(* PLC project NETWORK, CODESYS CODESYS V3.5 SP16, author OSCAT *)
(* stored: creationDateTime 2021-04-18T12:40:34.2115358, version 1.3.5.2, modificationDateTime 2021-03-02T15:47:52, organization OSCAT *)
(* Oscat Network Version 07/2017 aus *.lib
Formale Korrekturen von annD und Referenzen "Variabeln LOCAL_DT et.al." für Kompatibilität mit Codesys 3.5.16.0 und Oscat_Basic 3.3.4.0 angepasst *)

TYPE DLOG_CRON_DATA : STRUCT
  CE : ARRAY[0..5] OF DLOG_CRON_ELEMENT;
END_STRUCT;
END_TYPE

TYPE DLOG_CRON_ELEMENT : STRUCT
  ELEMENTS : ARRAY[0..59] OF BOOL;
  VALUE : INT;
  VALUE_MIN : INT;
  VALUE_MAX : INT;
  ALL_SELECTED : BOOL;
END_STRUCT;
END_TYPE

TYPE DLOG_DATA : STRUCT
  STORE_TYPE : BYTE;
  ADD_COM : INT;
  ADD_DATA_REQ : BOOL;
  CLOCK_TRIG : BOOL;
  ID_MAX : USINT;
  DTI : DT;
  UCB : UNI_CIRCULAR_BUFFER_DATA;
  LOAD_TIME_MAX : TIME;
  NEW_FILE : STRING;
  NEW_FILE_SIZE : UDINT;
  NEW_FILE_RTRIG : BOOL;
END_STRUCT;
END_TYPE

TYPE DLOG_REAL_ARRAY_DATA : ARRAY[1..64] OF DLOG_REAL_ARRAY_ELEMENT;
END_TYPE

TYPE DLOG_REAL_ARRAY_ELEMENT : STRUCT
  VALUE : REAL;
  DELTA : REAL;
  COLUMN : STRING(10);
  _DELTA_LAST : REAL;
  _VALUE_LAST : REAL;
END_STRUCT;
END_TYPE

TYPE DLOG_RETAIN : STRUCT
  FN_REM : STRING;
  COLOR : BOOL;
  HEAD : BOOL;
  TRIG_CNT : UDINT;
  TRIG_CNT_TOTAL : UDINT;
END_STRUCT;
END_TYPE

TYPE DLOG_SAVE : STRUCT
  FN_REM : STRING;
  COLOR : BOOL;
  HEAD : BOOL;
  TRIG_CNT : UDINT;
  TRIG_CNT_TOTAL : UDINT;
END_STRUCT;
END_TYPE

TYPE LOG_CONTROL : STRUCT
  NEW_MSG : STRING(LOG_SIZE);  (* neue Nachricht für den Datenbuffer *)
  NEW_MSG_OPTION : DWORD;
  LEVEL : BYTE;
  SIZE : INT := LOG_MAX;  (* Anzahl der Strings im LOG_DATA *)
  RESET : BOOL;  (* Nachrichtenbuffer löschen *)
  PRINTF : PRINTF_DATA;  (* Array PRINTF Parameter *)
  MSG : ARRAY[0..LOG_MAX] OF STRING(LOG_SIZE);  (* Array Message *)
  MSG_OPTION : ARRAY[0..LOG_MAX] OF DWORD;  (* Array Options *)
  UPDATE_COUNT : UINT;  (* Updatezähler *)
  IDX : INT;  (* aktueller Nachrichten-Index *)
  RING_MODE : BOOL;  (* Bufferüberlauf erkannt *)
END_STRUCT;
END_TYPE

TYPE PRINTF_DATA : ARRAY[1..11] OF STRING(LOG_SIZE);
END_TYPE

TYPE UNI_CIRCULAR_BUF : ARRAY[0..8191] OF BYTE;
END_TYPE

TYPE UNI_CIRCULAR_BUFFER_DATA : STRUCT
  D_MODE : INT;
  D_SIZE : INT;
  D_HEAD : WORD;
  D_STRING : STRING(OSCAT_BASIC.STRING_LENGTH);
  D_REAL : REAL;
  D_DWORD : DWORD;
  BUF_SIZE : UINT;
  BUF_COUNT : UINT;
  BUF_USED : USINT;
  BUF_USED_MAX : USINT;
  BUF_DATA_CNT : UDINT;
  BUF_DATA_LOST : UDINT;
  BUF : UNI_CIRCULAR_BUF;
  _GetStart : UINT;
  _GetEnd : UINT;
  _Last : UINT;
  _First : UINT;
END_STRUCT;
END_TYPE

TYPE us_LOG_VIEWPORT : STRUCT
  LINE_ARRAY : ARRAY[1..40] OF INT;
  COUNT : INT;  (* Anzahl der sichtbaren Nachtrichten *)
  UPDATE_COUNT : UINT;  (* Updatezähler *)
  MOVE_TO_X : INT;  (* Steuerung der Nachrichtenanzeige *)
  UPDATE : BOOL;  (* Daten wurden geändert -> neuzeichnen *)
END_STRUCT;
END_TYPE

TYPE MYSQL_COM : STRUCT
  S_BUF : NETWORK_BUFFER;
  R_BUF : NETWORK_BUFFER;
  SQL_CON : BOOL;
  SQL_URL : STRING(OSCAT_BASIC.STRING_LENGTH);
  SQL_PACKET_NO : BYTE;
  TIMEOUT : TIME;
  DNS_IP4 : DWORD;
  SQL_RCV_STATE : BYTE;
  ERROR_C : DWORD;
  ERROR_T : BYTE;
END_STRUCT;
END_TYPE

TYPE MYSQL_INFO : STRUCT
  SERVER_PROTOCOL_VERSION : BYTE;
  SERVER_CAPABILITIES : WORD;
  SERVER_STATUS : WORD;
  SERVER_LANGUAGE : BYTE;
  SQL_CONNECTED : BOOL;
  SQL_ERROR : STRING(OSCAT_BASIC.STRING_LENGTH);
  DATA_INSERT_AKTIV : BOOL;
  DATA_INSERT_OK_CNT : UDINT;
  DATA_INSERT_NOK_CNT : UDINT;
END_STRUCT;
END_TYPE

TYPE FILE_PATH_DATA : STRUCT
  DRIVE : STRING(3);
  DIRECTORY : STRING(OSCAT_BASIC.STRING_LENGTH);
  FILENAME : STRING;
END_STRUCT;
END_TYPE

TYPE FILE_SERVER_DATA : STRUCT
  FILE_OPEN : BOOL;
  FILENAME : STRING;
  MODE : BYTE;
  OFFSET : UDINT;
  FILE_SIZE : UDINT;
  ERROR : BYTE;
  RUNTIME : FILE_SERVER_RUNTIME_DATA;
END_STRUCT;
END_TYPE

TYPE FILE_SERVER_RUNTIME_DATA : STRUCT
  TIME_FILE_OPEN_CUR : UDINT;
  TIME_FILE_OPEN_MAX : UDINT;
  TIME_FILE_OPEN_MIN : UDINT;
  TIME_FILE_CLOSE_CUR : UDINT;
  TIME_FILE_CLOSE_MAX : UDINT;
  TIME_FILE_CLOSE_MIN : UDINT;
  TIME_FILE_READ_CUR : UDINT;
  TIME_FILE_READ_MAX : UDINT;
  TIME_FILE_READ_MIN : UDINT;
  TIME_FILE_WRITE_CUR : UDINT;
  TIME_FILE_WRITE_MAX : UDINT;
  TIME_FILE_WRITE_MIN : UDINT;
  TIME_FILE_SEEK_CUR : UDINT;
  TIME_FILE_SEEK_MAX : UDINT;
  TIME_FILE_SEEK_MIN : UDINT;
  TIME_FILE_TELL_CUR : UDINT;
  TIME_FILE_TELL_MAX : UDINT;
  TIME_FILE_TELL_MIN : UDINT;
  TIME_FILE_DELETE_CUR : UDINT;
  TIME_FILE_DELETE_MAX : UDINT;
  TIME_FILE_DELETE_MIN : UDINT;
END_STRUCT;
END_TYPE

TYPE NET_VAR_DATA : STRUCT
  CYCLE : UDINT;
  STATE : BYTE;
  INDEX : INT;
  ID_MAX : USINT;
  ERROR_ID : BYTE;
  BUF_SIZE : UINT;
  S_BUF : NETWORK_BUFFER;
  R_BUF : NETWORK_BUFFER;
END_STRUCT;
END_TYPE

TYPE IP_C : STRUCT
  C_MODE : BYTE;  (* W Mode: TCP/UCP AKTIV/PASSIV *)
  C_PORT : WORD;  (* W Portnummer *)
  C_IP : DWORD;  (* W IP-Adresse gepackt wwxxyyzz = www.xxx.yyy.zzz *)
  C_STATE : BYTE;  (* R Verbindungsstatus ON/OFF + Flanke ON/OFF *)
  C_ENABLE : BOOL;  (* W Freigabe für Connect *)
  R_OBSERVE : BOOL;  (* W Empfang ueberwachen *)
  TIME_RESET : BOOL;  (* W Alle Timer ruecksetzen *)
  ERROR : DWORD;  (* R vvwwxxyy (vv = CON_ERROR, ww = SEN_ERROR, xx = REC_ERROR *)
  FIFO : IP_FIFO_DATA;  (* I IP FIFO Struktur *)
  MAILBOX : ARRAY[1..16] OF BYTE;  (* I Mailbox: Datenbereich für Bausteindatenaustausch *)
END_STRUCT;
END_TYPE

TYPE IP_FIFO_DATA : STRUCT
  X : ARRAY[1..128] OF BYTE;  (* IP_ID FIFO Speicher *)
  Y : ARRAY[1..128] OF BYTE;  (* IP_ID Zähler *)
  ID : BYTE;  (* höchste vergabene id *)
  MAX_ID : BYTE;  (* maximal Anmeldungen pro ID *)
  INIT : BOOL;  (* Initialisierung durchgeführt *)
  EMPTY : BOOL;  (* FIFO leer *)
  FULL : BOOL;  (* FIFO voll *)
  TOP : INT;  (* maximale anzahl in FIFO *)
  NW : INT;  (* Schreibzeiger *)
  NR : INT;  (* Lesezeiger *)
END_STRUCT;
END_TYPE

TYPE IP2GEO_DATA : STRUCT
  STATE : BOOL;
  IP4 : DWORD;
  COUNTRY_CODE : STRING(2);
  COUNTRY_NAME : STRING(20);
  REGION_CODE : STRING(2);
  REGION_NAME : STRING(20);
  CITY : STRING(20);
  GEO_LATITUDE : REAL;
  GEO_LONGITUDE : REAL;
  TIME_ZONE_NAME : STRING(20);
  GMT_OFFSET : INT;
  IS_DST : BOOL;
END_STRUCT;
END_TYPE

TYPE NETWORK_BUFFER : STRUCT
  SIZE : UINT;
  BUFFER : NW_BUF_LONG;
END_STRUCT;
END_TYPE

TYPE NETWORK_BUFFER_SHORT : STRUCT
  SIZE : UINT;
  BUFFER : NW_BUF_SHORT;
END_STRUCT;
END_TYPE

TYPE NW_BUF_LONG : ARRAY[0..NETWORK_BUFFER_LONG_SIZE] OF BYTE;
END_TYPE

TYPE NW_BUF_SHORT : ARRAY[0..NETWORK_BUFFER_SHORT_SIZE] OF BYTE;
END_TYPE

TYPE URL : STRUCT
  PROTOCOL : STRING(10);
  USER : STRING(32);
  PASSWORD : STRING(32);
  DOMAIN : STRING(80);
  PORT : WORD;
  PATH : STRING(80);
  QUERY : STRING(OSCAT_BASIC.STRING_LENGTH);
  ANCHOR : STRING(40);
  HEADER : STRING(160);
END_STRUCT;
END_TYPE

TYPE VMAP_DATA : STRUCT
  FC : DWORD;
  V_ADR : INT;
  V_SIZE : INT;
  P_ADR : INT;
  TIME_OUT : TIME;
END_STRUCT;
END_TYPE

TYPE XML_CONTROL : STRUCT
  COMMAND : WORD;
  WATCHDOG : TIME;
  START_POS : UINT;
  STOP_POS : UINT;
  COUNT : UINT;
  TYP : INT;
  LEVEL : UINT;
  PATH : STRING(OSCAT_BASIC.STRING_LENGTH);
  ELEMENT : STRING(OSCAT_BASIC.STRING_LENGTH);
  ATTRIBUTE : STRING(OSCAT_BASIC.STRING_LENGTH);
  VALUE : STRING(OSCAT_BASIC.STRING_LENGTH);
  BLOCK1_START : UINT;
  BLOCK1_STOP : UINT;
  BLOCK2_START : UINT;
  BLOCK2_STOP : UINT;
END_STRUCT;
END_TYPE

TYPE us_TN_INPUT_CONTROL : STRUCT
  bo_Enable : BOOL;  (* Bearbeitung freigeben/sperren *)
  bo_Update_all : BOOL;  (* All Elemente neu zeichnen *)
  bo_Reset_Fokus : BOOL;  (* Fokus auf 1. Element setzen *)
  in_Focus_at : INT;  (* Controlelement mit aktivem Fokus *)
  in_Count : INT;  (* Anzahl der benutzen Control-Elemente *)
  in_ToolTip_X : INT;  (* Tooltip Text X-Offset *)
  in_ToolTip_Y : INT;  (* Tooltip Text Y-Offset *)
  by_ToolTip_Attr : BYTE;  (* Tooltip Text Attribute *)
  in_ToolTip_Size : INT;  (* Tooltip Text länge *)
  usa_TN_INPUT_CONTROL_DATA : ARRAY[1..20] OF us_TN_INPUT_CONTROL_DATA;
END_STRUCT;
END_TYPE

TYPE us_TN_INPUT_CONTROL_DATA : STRUCT
  by_Input_Exten_Code : BYTE;
  by_Input_ASCII_Code : BYTE;
  bo_Input_ASCII_IsNum : BOOL;
  in_Title_X_Offset : INT;  (* Title Text X-Offset *)
  in_Title_Y_Offset : INT;  (* Title Text Y-Offset *)
  by_Title_Attr : BYTE;  (* Title Text Attribute *)
  st_Title_String : STRING;  (* Title Text String *)
  in_Cursor_X : INT;  (* aktuelle Cursor X-Position *)
  in_Cursor_Y : INT;  (* aktuelle Cursor Y-Position *)
  in_Type : INT;  (* Type des Elements *)
  in_X : INT;  (* Element X-Position *)
  in_Y : INT;  (* Element Y-Position *)
  in_Cursor_Pos : INT;  (* aktuelle Cursorposition *)
  by_Attr_mF : BYTE;  (* Text Attribute mit Fokus *)
  by_Attr_oF : BYTE;  (* Text Attribute ohne Fokus *)
  in_selected : INT;  (* Text Item wurde ausgewählt *)
  st_Input_Mask : STRING;  (* Text Eingabemaske *)
  st_Input_Data : STRING(OSCAT_BASIC.STRING_LENGTH);  (* Text aktuelle Eingabedaten *)
  st_Input_String : STRING;  (* Text Kopie nach Return-Taste *)
  st_Input_ToolTip : STRING;  (* Text ToolTip (Eingabeinformation) *)
  in_Input_Option : INT;  (* Text Ausgabe-Optionen *)
  bo_Input_Entered : BOOL;  (* RETURN-Taste wurde betätigt *)
  bo_Input_Hidden : BOOL;  (* Text versteckete Eingabe mit '*' *)
  bo_Input_Only_Num : BOOL;  (* Text nur Nummerneingabe zulassen *)
  bo_Focus : BOOL;  (* Element besitzt den Fokus *)
  bo_Update_Input : BOOL;  (* Element wegen Benutzereingabe neuzeichnen *)
  bo_Update_All : BOOL;  (* Element komplett neuzeichnen *)
END_STRUCT;
END_TYPE

TYPE us_TN_MENU : STRUCT
  st_Menu_Text : STRING(OSCAT_BASIC.STRING_LENGTH);  (* X Menue Texte *)
  in_Menu_E_Count : INT;  (* Menue Elemente Anzahl *)
  in_Y : INT;  (* Menue Zeilennummer Y-Position *)
  in_X : INT;  (* Menue Spaltennummer X-Position *)
  by_Attr_mF : BYTE;  (* Text Attribute mit Fokus *)
  by_Attr_oF : BYTE;  (* Text Attribute ohne Fokus *)
  in_X_SM_new : INT;  (* neue Sub-Menu X-Position *)
  in_Y_SM_new : INT;  (* neue Sub-Menu Y-Position *)
  in_X_SM_old : INT;  (* alte Sub-Menu X-Position *)
  in_Y_SM_old : INT;  (* alte Sub-Menu Y-Position *)
  in_Cur_Menu_Item : INT;  (* aktuelles Haupt-Menue *)
  in_Cur_Sub_Item : INT;  (* aktuelles Sub-Menue *)
  in_State : INT;  (* Menu status *)
  in_Menu_Selected : INT;  (* X Menu-Item mit Enter angewwählt *)
  bo_Create : BOOL;  (* X Menu erzeugen *)
  bo_Destroy : BOOL;  (* X Menu entfernen *)
  bo_Update : BOOL;  (* X Menu updaten *)
END_STRUCT;
END_TYPE

TYPE us_TN_MENU_POPUP : STRUCT
  st_Menu_Text : STRING(OSCAT_BASIC.STRING_LENGTH);  (* X Menue Texte *)
  in_Menu_E_Count : INT;  (* Menue Elemente Anzahl *)
  in_X : INT;  (* X Menue X-Position *)
  in_Y : INT;  (* X Menue Y-Position *)
  in_Cols : INT;  (* Menue Spaltenanzahl *)
  in_Rows : INT;  (* Menue Zeilenanzahl *)
  in_Cur_Item : INT;  (* X aktuelles Sub-Menue *)
  by_Attr_mF : BYTE;  (* X Text Attribute mit Fokus *)
  by_Attr_oF : BYTE;  (* X Text Attribute ohne Fokus *)
  by_Input_Exten_Code : BYTE;  (* X Tastencode: Sondertasten *)
  bo_Create : BOOL;  (* X Popup-Menu erzeugen *)
  bo_Destroy : BOOL;  (* X Popup-Menu entfernen *)
  bo_Update : BOOL;  (* X Popup-Menu updaten *)
  bo_Activ : BOOL;  (* Popup-Menu ist aktiv *)
END_STRUCT;
END_TYPE

TYPE us_TN_SCREEN : STRUCT
  bya_CHAR : ARRAY[0..1919] OF BYTE;
  bya_COLOR : ARRAY[0..1919] OF BYTE;
  bya_BACKUP : ARRAY[0..1919] OF BYTE;
  bya_Line_Update : ARRAY[0..23] OF BOOL;
  by_Input_Exten_Code : BYTE;
  by_Input_ASCII_Code : BYTE;
  bo_Input_ASCII_IsNum : BOOL;
  in_Page_Number : INT;  (* aktive Seiten-Nr. *)
  in_Cursor_X : INT;  (* Cursor X-Position *)
  in_Cursor_Y : INT;  (* Cursor Y-Position *)
  in_EOS_Offset : INT;  (* End of String Offset *)
  by_Clear_Screen_Attr : BYTE;  (* Clear-Screen Attr *)
  bo_Clear_Screen : BOOL;  (* Clear-Screen auslösen *)
  bo_Modal_Dialog : BOOL;  (* Modaler Dialog ist aktiv *)
  bo_Menue_Bar_Dialog : BOOL;  (* Menue Dialog ist aktiv *)
END_STRUCT;
END_TYPE

TYPE WORLD_WEATHER_CUR : STRUCT
  OBSERVATION_TIME : STRING(8);
  TEMP_C : INT;
  WEATHER_CODE : INT;
  WEATHER_DESC : STRING(60);
  WEATHER_ICON : INT;
  WIND_SPEED_MILES : INT;
  WIND_SPEED_KMPH : INT;
  WIND_DIR_DEGREE : INT;
  WIND_DIR16POINT : STRING(3);
  PRECIPMM : REAL;
  HUMIDITY : INT;
  VISIBILITY : INT;
  PRESSURE : INT;
  CLOUDOVER : INT;
END_STRUCT;
END_TYPE

TYPE WORLD_WEATHER_DATA : STRUCT
  CUR : WORLD_WEATHER_CUR;
  DAY : ARRAY[0..4] OF WORLD_WEATHER_DAY;
END_STRUCT;
END_TYPE

TYPE WORLD_WEATHER_DAY : STRUCT
  DATE_OF_DAY : STRING(10);
  TEMP_MAX_C : INT;
  TEMP_MAX_F : INT;
  TEMP_MIN_C : INT;
  TEMP_MIN_F : INT;
  WIND_SPEED_MILES : INT;
  WIND_SPEED_KMPH : INT;
  WIND_DIR_DEGREE : INT;
  WIND_DIR16POINT : STRING(3);
  WEATHER_CODE : INT;
  WEATHER_DESC : STRING(60);
  WEATHER_ICON : INT;
  PRECIPMM : REAL;
END_STRUCT;
END_TYPE

TYPE YAHOO_WEATHER_DATA : STRUCT
  LOCATION_CITY : STRING(40);  (* THE LOCATION OF THIS FORECAST: CITY: CITY NAME *)
  LOCATION_REGION : STRING(20);  (* THE LOCATION OF THIS FORECAST: REGION: STATE, TERRITORY, OR REGION, IF GIVEN *)
  LOCATION_COUNTRY : STRING(20);  (* THE LOCATION OF THIS FORECAST: COUNTRY: TWO-CHARACTER COUNTRY CODE *)
  UNIT_TEMPERATURE : STRING(1);  (* TEMPERATURE: DEGREE UNITS, F FOR FAHRENHEIT OR C FOR CELSIUS *)
  UNIT_DISTANCE : STRING(2);  (* DISTANCE: UNITS FOR DISTANCE, MI FOR MILES OR KM FOR KILOMETERS *)
  UNIT_PRESSURE : STRING(2);  (* PRESSURE: UNITS OF BAROMETRIC PRESSURE, IN FOR POUNDS PER SQUARE INCH OR MB FOR MILLIBARS *)
  UNIT_SPEED : STRING(4);  (* SPEED: UNITS OF SPEED, MPH FOR MILES PER HOUR OR KPH FOR KILOMETERS PER HOUR *)
  WIND_CHILL : INT;  (* FORECAST INFORMATION ABOUT WIND CHILL IN DEGREES *)
  WIND_DIRECTION : INT;  (* FORECAST INFORMATION ABOUT WIND DIRECTION, IN DEGREES *)
  WIND_SPEED : REAL;  (* FORECAST INFORMATION ABOUT WIND SPEED, IN THE UNITS (MPH OR KPH) *)
  ATMOSPHERE_HUMIDITY : INT;  (* FORECAST INFORMATION ABOUT CURRENT ATMOSPHERIC HUMIDITY: HUMIDITY, IN PERCENT *)
  ATMOSPHERE_PRESSURE : REAL;  (* FORECAST INFORMATION ABOUT CURRENT ATMOSPHERIC PRESSURE: BAROMETRIC PRESSURE, IN THE UNITS (IN OR MB) *)
  ATMOSPHERE_VISIBILITY : REAL;  (* FORECAST INFORMATION ABOUT CURRENT ATMOSPHERIC VISIBILITY, IN THE UNITS (MI OR KM) *)
  ATMOSPHERE_RISING : INT;  (* FORECAST INFORMATION ABOUT RISING: STATE OF THE BAROMETRIC PRESSURE: STEADY (0), RISING (1), OR FALLING (2). (INTEGER: 0, 1, 2) *)
  ASTRONOMY_SUNRISE : STRING(10);  (* SUNRISE: TODAY'S SUNRISE TIME. THE TIME IS A STRING IN A LOCAL TIME FORMAT OF "H:MM AM/PM" *)
  ASTRONOMY_SUNSET : STRING(10);  (* SUNSET: TODAY'S SUNSET TIME. THE TIME IS A STRING IN A LOCAL TIME FORMAT OF "H:MM AM/PM", *)
  GEO_LATITUDE : REAL;  (* THE LATITUDE OF THE LOCATION *)
  GEO_LONGITUDE : REAL;  (* THE LONGITUDE OF THE LOCATION *)
  CUR_CONDITIONS_TEMP : INT;  (* THE CURRENT WEATHER CONDITIONS: TEMP: THE CURRENT TEMPERATURE, IN THE UNITS (F OR C) *)
  CUR_CONDITIONS_TEXT : STRING(40);  (* THE CURRENT WEATHER CONDITIONS: TEXT: A TEXTUAL DESCRIPTION OF CONDITIONS *)
  CUR_CONDITIONS_CODE : INT;  (* THE CURRENT WEATHER CONDITIONS: CODE: THE CONDITION CODE FOR THIS FORECAST *)
  CUR_CONDITIONS_ICON : INT;  (* THE CURRENT WEATHER CONDITIONS: ICON: THE CONDITION ICON FOR THIS FORECAST *)
  FORECAST_TODAY_LOW_TEMP : INT;  (* THE FORECAST TODAY WEATHER CONDITIONS: THE FORECASTED LOW TEMPERATURE FOR THIS DAY IN THE UNITS (F OR C) *)
  FORECAST_TODAY_HIGH_TEMP : INT;  (* THE FORECAST TODAY WEATHER CONDITIONS: THE FORECASTED HIGH TEMPERATURE FOR THIS DAY IN THE UNITS (F OR C) *)
  FORECAST_TODAY_TEXT : STRING(40);  (* THE FORECAST TODAY WEATHER CONDITIONS: TEXT: A TEXTUAL DESCRIPTION OF CONDITIONS *)
  FORECAST_TODAY_CODE : INT;  (* THE CURRENT WEATHER CONDITIONS: CODE: THE CONDITION CODE FOR THIS FORECAST *)
  FORECAST_TODAY_ICON : INT;  (* THE CURRENT WEATHER CONDITIONS: ICON: THE CONDITION ICON FOR THIS FORECAST *)
  FORECAST_TODAY_DATE_LONG : STRING(20);  (* THE CURRENT WEATHER CONDITIONS: DATE: DATE OF THE DAY *)
  FORECAST_DAY : ARRAY[1..9] OF YAHOO_WEATHER_FORECAST_DAY;  (* THE CURRENT WEATHER DAYS ARRAY *)
END_STRUCT;
END_TYPE

TYPE YAHOO_WEATHER_FORECAST_DAY : STRUCT
  LOW_TEMP : INT;  (* THE FORECAST WEATHER CONDITIONS: THE FORECASTED LOW TEMPERATURE FOR THIS DAY IN THE UNITS (F OR C) *)
  HIGH_TEMP : INT;  (* THE FORECAST WEATHER CONDITIONS: THE FORECASTED HIGH TEMPERATURE FOR THIS DAY IN THE UNITS (F OR C) *)
  TEXT : STRING(40);  (* THE FORECAST WEATHER CONDITIONS: TEXT: A TEXTUAL DESCRIPTION OF CONDITIONS *)
  DATE_LONG : STRING(20);  (* THE FORECAST WEATHER CONDITIONS: DATE: DATE OF THE DAY *)
  CODE : INT;  (* THE FORECAST WEATHER CONDITIONS: CODE: THE CONDITION CODE FOR THIS FORECAST *)
  ICON : INT;  (* THE FORECAST WEATHER CONDITIONS: ICON: THE CONDITION ICON FOR THIS FORECAST *)
END_STRUCT;
END_TYPE

VAR_GLOBAL CONSTANT  (* Constants *)
  NETWORK_BUFFER_LONG_SIZE : UINT := 4095;
  NETWORK_BUFFER_SHORT_SIZE : UINT := 1407;
  LOG_MAX : INT := 40;
  LOG_SIZE : INT := 80;
  ELEMENT_LENGTH : INT := 250;
END_VAR

VAR_GLOBAL  (* Globale_Variablen *)
  TCP_SERVER_RESET : BYTE;  (* only for internaly use - do't modify *)
  sSrvNetId : STRING(23) := '';  (* String containing the network address of the TwinCAT TCP/IP Connection Server (e.g. '1.1.1.2.7.1'). For the local computer (default) an empty string may be specified *)
  sLocalHost : STRING(15) := '';  (* The local IP address (Ipv4) of the UDP client/server socket as a string (e.g. '172.33.5.1'). An empty string may be specified for the default network adapter *)
  SYSLIBSOCKETS_OPTION : BYTE := BYTE#16#0;  (* --------------------------------------------- ------- only for CoDeSys -------------------- Configuration for SysLibSocket.lib Bit 0 = 1 -> PLCWinNT Bit 1 = 1 -> PLC WAGO 750-841 Bit 2 = 1 -> PLC WAGO 750-881 *)
  LOG_CL : LOG_CONTROL;  (* ---------------------------------------------------- *)
END_VAR

FUNCTION_BLOCK BASE64_DECODE_STR
  VAR_INPUT
    RUN : BOOL;
  END_VAR
  VAR_OUTPUT
    DONE : BOOL;
  END_VAR
  VAR_IN_OUT
    STR1 : STRING(192);
    STR2 : STRING(144);
  END_VAR
  VAR
    BASE64_DECODE_STREAM : BASE64_DECODE_STREAM;
    run_last : BOOL;
    buf1 : ARRAY[0..63] OF BYTE;
    buf2 : ARRAY[0..47] OF BYTE;
    mode : INT;
    size1 : INT;
    size2 : INT;
    end : INT;
    pos : INT;
  END_VAR

            CASE mode OF
0:	IF RUN AND NOT run_last THEN
		DONE := FALSE;
		mode := 1;
		end := LEN(STR1);
		pos := 0;
		STR2 := '';
	END_IF;
1:
	size1 := MIN(48,end - pos);
	IF size1 > 0 THEN
		OSCAT_BASIC._STRING_TO_BUFFER(STR:=MID(STR1, size1, pos + 1), POS:=0, PT:=ADR(buf1), SIZE:=SIZEOF(buf1));
		BASE64_DECODE_STREAM(BUF1:=buf1 ,BUF2:=buf2 ,SIZE1:=size1 ,SIZE2=>size2);
		STR2 := CONCAT(STR2,OSCAT_BASIC.BUFFER_TO_STRING(PT:=ADR(buf2), SIZE:=SIZEOF(buf2), START:=0, STOP:=size2 - 1));
	ELSE
		mode := 0;
		DONE := TRUE;
	END_IF;
	pos := pos + size1;
END_CASE;

run_last := RUN;

(* revision history

ks	6. dec. 2009 rev 1.0
	original version

*)
          
END_FUNCTION_BLOCK

FUNCTION_BLOCK BASE64_DECODE_STREAM
  VAR_IN_OUT
    BUF1 : ARRAY[0..63] OF BYTE;
    BUF2 : ARRAY[0..47] OF BYTE;
  END_VAR
  VAR_INPUT
    SIZE1 : INT;
  END_VAR
  VAR_OUTPUT
    SIZE2 : INT;
  END_VAR
  VAR_TEMP
    a : INT;
    b : WORD;
    o : INT;
    off : INT;
    i1 : INT;
    i2 : INT;
    c : INT;
  END_VAR

            IF SIZE1 <= 0 THEN SIZE2 := 0; RETURN; END_IF;
c := SIZE1 - 1;
i2 := 0;
a := 0;
b := 0;
FOR i1 := 0 TO c DO
	o := BUF1[i1];
	IF o = 61  (* = *) THEN	EXIT;
	ELSIF o > 96 (* a-z *) THEN off := 71;
	ELSIF o > 64 (* A-Z *) THEN off := 65;
	ELSIF o > 47 (* 0-9 *) THEN off := -4;
	ELSIF o = 43 (* + *) THEN off := -19;
	ELSIF o = 47 (* / *) THEN off := -16;
	END_IF;
	b := SHL(b,6) OR INT_TO_BYTE(o - off);
	a := a + 6;
	IF a >= 8 THEN
		a := a - 8;
		BUF2[i2] := WORD_TO_BYTE(SHR(b,a));
		i2 := i2 + 1;
		b := b AND NOT SHL(WORD#16#FFFF,a);
	END_IF;
END_FOR;
SIZE2 := i2;

(* revision history

ks	6. dec. 2009 rev 1.0
	original version

*)
          
END_FUNCTION_BLOCK

FUNCTION_BLOCK BASE64_ENCODE_STR
  VAR_INPUT
    RUN : BOOL;
  END_VAR
  VAR_OUTPUT
    DONE : BOOL;
  END_VAR
  VAR_IN_OUT
    STR1 : STRING(144);
    STR2 : STRING(192);
  END_VAR
  VAR
    BASE64_ENCODE_STREAM : BASE64_ENCODE_STREAM;
    run_last : BOOL;
    buf1 : ARRAY[0..47] OF BYTE;
    buf2 : ARRAY[0..63] OF BYTE;
    mode : INT;
    size1 : INT;
    size2 : INT;
    end : INT;
    pos : INT;
  END_VAR

            CASE mode OF
0:	IF RUN AND NOT run_last THEN
		DONE := FALSE;
		mode := 1;
		end := LEN(STR1);
		pos := 0;
		STR2 := '';
	END_IF;
1:
	size1 := MIN(48,end - pos);
	IF size1 > 0 THEN
		OSCAT_BASIC._STRING_TO_BUFFER(STR:=MID(STR1, size1, pos + 1), POS:=0, PT:=ADR(buf1), SIZE:=SIZEOF(buf1));
		BASE64_ENCODE_STREAM(BUF1:=buf1 ,BUF2:=buf2 ,SIZE1:=size1 ,SIZE2=>size2);
		STR2 := CONCAT(STR2,OSCAT_BASIC.BUFFER_TO_STRING(PT:=ADR(buf2), SIZE:=SIZEOF(buf2), START:=0, STOP:=size2 - 1));
	ELSE
		mode := 0;
		DONE := TRUE;
	END_IF;
	pos := pos + size1;
END_CASE;

run_last := RUN;

(* revision history

ks	6. dec. 2009 rev 1.0
	original version

*)
          
END_FUNCTION_BLOCK

FUNCTION_BLOCK BASE64_ENCODE_STREAM
  VAR_IN_OUT
    BUF1 : ARRAY[0..47] OF BYTE;
    BUF2 : ARRAY[0..63] OF BYTE;
  END_VAR
  VAR_INPUT
    SIZE1 : INT;
  END_VAR
  VAR_OUTPUT
    SIZE2 : INT;
  END_VAR
  VAR
    a : INT;
    b : WORD;
    i : INT;
    i2 : INT;
    i3 : INT;
    c : INT;
    BASE64 : STRING(64) := 'ABCDEFGHIJKLMNOPQRSTUVWXYZabcdefghijklmnopqrstuvwxyz0123456789+/';
  END_VAR

            IF SIZE1 <= 0 THEN
	SIZE2 := 0;
	RETURN;
END_IF;
c := SIZE1 - 1;
i2 := 0;
a := 0;
b := 0;
FOR i := 0 TO c DO
	b := SHL(b,8) OR BUF1[i];
	a := a + 8;
	WHILE a >= 6 DO
		a := a - 6;
		buf2[i2] := OSCAT_BASIC.CODE(BASE64,WORD_TO_INT(SHR(b,a)) + 1);
		i2 := i2 + 1;
		b := b AND NOT SHL(WORD#16#FFFF,a);
	END_WHILE;
END_FOR;
IF a > 0 THEN
	buf2[i2] := OSCAT_BASIC.CODE(BASE64,WORD_TO_INT(SHL(b,6 - a)) + 1);
	i2 := i2 + 1;
	i3 := i2 + (NOT INT_TO_WORD(i2) AND 2#11);
	FOR i := i2 TO i3 DO
		buf2[i] := 61;
	END_FOR;
	SIZE2 := i3 + 1;
ELSE
	SIZE2 := i2;
END_IF;

(* revision history

ks	6. dec. 2009 rev 1.0
	original version

*)
          
END_FUNCTION_BLOCK

FUNCTION HTML_DECODE : STRING(OSCAT_BASIC.STRING_LENGTH)
  VAR_INPUT
    IN : STRING(OSCAT_BASIC.STRING_LENGTH);
  END_VAR
  VAR
    pos : INT;
    end : INT;
    tmp : STRING(10);
    code : STRING(1);
  END_VAR

            HTML_DECODE := IN;

(* docode characters encoded by character position *)
pos := FIND(HTML_DECODE, '&');
WHILE pos > 0 DO
	tmp := MID(HTML_DECODE, 2, pos + 1);
	IF tmp = '#x' OR tmp = '#X' THEN
		(* hexadecimal representation found *)
		tmp := MID(HTML_DECODE, 10, pos + 3);
		end := FIND(tmp, ';');
		CODE := OSCAT_BASIC.CHR_TO_STRING(DWORD_TO_BYTE(OSCAT_BASIC.HEX_TO_DWORD(LEFT(tmp, end - 1))));
		HTML_DECODE := REPLACE(HTML_DECODE, CODE, end + 3, pos);
	ELSIF LEFT(tmp,1) = '#' THEN
		tmp := MID(HTML_DECODE, 10, pos + 2);
		end := FIND(tmp, ';');
		CODE := OSCAT_BASIC.CHR_TO_STRING(INT_TO_BYTE(STRING_TO_INT(LEFT(tmp, end - 1))));
		HTML_DECODE := REPLACE(HTML_DECODE, CODE, end + 2, pos);
	ELSE
		(* replace all named characters *)
		tmp := MID(HTML_DECODE, 10, pos + 1);
		end := FIND(tmp, ';');
		CODE := OSCAT_BASIC.CHR_TO_STRING(OSCAT_BASIC.CHARCODE(LEFT(tmp, end - 1)));
		HTML_DECODE := REPLACE(HTML_DECODE, CODE, end + 1, pos);
	END_IF;
	(* search for next occurence of encoded characters *)
	pos := OSCAT_BASIC.FINDP(HTML_DECODE, '&', pos + 1);
END_WHILE;



(* revision history
hm	3. mai. 2008	rev 1.0
	original version

hm	16. jun. 2008	rev 1.1
	changed nested call of replace for better compatibility

hm	17. dec. 2008	rev 1.2
	changed function CHR to CHR_TO_STRING

hm	10. may. 2010	rev 1.3
	stringlength 250

*)
          
END_FUNCTION

FUNCTION HTML_ENCODE : STRING(OSCAT_BASIC.STRING_LENGTH)
  VAR_INPUT
    IN : STRING(OSCAT_BASIC.STRING_LENGTH);
    M : BOOL;
  END_VAR
  VAR
    pt_in : POINTER TO ARRAY[1..255] OF BYTE;
    pt_out : POINTER TO ARRAY[1..256] OF BYTE;
    pos_in : INT;
    pos_out : INT;
    stop : INT;
    B : BYTE;
    tmp : STRING(10);
    i : INT;
  END_VAR

            pt_in  := ADR(in);
pt_out := ADR(HTML_ENCODE);

(* scan the input string and convert unallowed characters *)
pos_in := 1;
stop := LEN(in);
FOR pos_out := 1 TO 250 DO
	IF pos_in > stop THEN EXIT; END_IF;
	B := pt_in^[pos_in];
	CASE BYTE_TO_INT(B) OF
		34: (* " detected *)
			IF pos_out > OSCAT_BASIC.STRING_LENGTH - 6 THEN EXIT; END_IF;
			pt_out^[pos_out] := 38;
			pos_out := pos_out + 1;
			pt_out^[pos_out] := 113;
			pos_out := pos_out + 1;
			pt_out^[pos_out] := 117;
			pos_out := pos_out + 1;
			pt_out^[pos_out] := 111;
			pos_out := pos_out + 1;
			pt_out^[pos_out] := 116;
			pos_out := pos_out + 1;
			pt_out^[pos_out] := 59;
		38: (* & detected *)
			IF pos_out > OSCAT_BASIC.STRING_LENGTH - 5 THEN EXIT; END_IF;
			pt_out^[pos_out] := 38;
			pos_out := pos_out + 1;
			pt_out^[pos_out] := 97;
			pos_out := pos_out + 1;
			pt_out^[pos_out] := 109;
			pos_out := pos_out + 1;
			pt_out^[pos_out] := 112;
			pos_out := pos_out + 1;
			pt_out^[pos_out] := 59;
		60: (* < detected *)
			IF pos_out > OSCAT_BASIC.STRING_LENGTH - 4 THEN EXIT; END_IF;
			pt_out^[pos_out] := 38;
			pos_out := pos_out + 1;
			pt_out^[pos_out] := 108;
			pos_out := pos_out + 1;
			pt_out^[pos_out] := 116;
			pos_out := pos_out + 1;
			pt_out^[pos_out] := 59;
		62: (* > detected *)
			IF pos_out > OSCAT_BASIC.STRING_LENGTH - 4 THEN EXIT; END_IF;
			pt_out^[pos_out] := 38;
			pos_out := pos_out + 1;
			pt_out^[pos_out] := 103;
			pos_out := pos_out + 1;
			pt_out^[pos_out] := 116;
			pos_out := pos_out + 1;
			pt_out^[pos_out] := 59;
	ELSE
		IF M AND B > 127 THEN
			tmp := OSCAT_BASIC.CHARNAME(B);
			(* exit if output string has not enough space *)
			IF pos_out + LEN(tmp) + 2 <= 250 THEN
				pt_out^[pos_out] := 38;
				pos_out := pos_out + 1;
				FOR i := 1 TO LEN(tmp) DO
					pt_out^[pos_out] := OSCAT_BASIC.CODE(tmp, i);
					pos_out := pos_out + 1;
				END_FOR;
				pt_out^[pos_out] := 59;
			END_IF;
		ELSE
			pt_out^[pos_out] := B;
		END_IF;
	END_CASE;
	(* increment in by 1 *)
	pos_in := pos_in + 1;
END_FOR;

(* terminate the output string *)
pt_out^[pos_out] := 0;



(* revision history
hm		3. mai. 2008	rev 1.0
	original version

hm		10. mai. 2008	rev 1.1
	stringlength 250
*)
          
END_FUNCTION

FUNCTION IP4_CHECK : BOOL
  VAR_INPUT
    NIP : DWORD;
    LIP : DWORD;
    SM : DWORD;
  END_VAR

            IP4_CHECK := (NIP AND sm) = (LIP AND SM);


(* revision history
hm		4. mar 2008	rev 1.0
	original version

*)
          
END_FUNCTION

FUNCTION IP4_DECODE : DWORD
  VAR_INPUT
    str : STRING(15);
  END_VAR
  VAR
    pos : INT;
  END_VAR

            pos := FIND(str, '.');
WHILE pos > 0 DO
	IP4_DECODE := SHL(IP4_DECODE,8) OR STRING_TO_DWORD(LEFT(str,pos - 1));
	str := DELETE(str, pos, 1);
	pos := FIND(str, '.');
END_WHILE;
IP4_DECODE := SHL(IP4_DECODE,8) OR STRING_TO_DWORD(str);


(* revision history
hm		29. feb 2008	rev 1.0
	original version

hm	10. mar. 2009	rev 1.1
	new algorythm
*)
          
END_FUNCTION

FUNCTION IP4_TO_STRING : STRING(15)
  VAR_INPUT
    IP4 : DWORD;
  END_VAR
  VAR
    tmp : STRING(3);
  END_VAR

            (* mask bits AND INSERT AT given position *)
tmp := BYTE_TO_STRING(DWORD_TO_BYTE(IP4));
IP4_TO_STRING := CONCAT('...', tmp);
tmp := BYTE_TO_STRING(DWORD_TO_BYTE(SHR(IP4,8)));
IP4_TO_STRING := INSERT(IP4_TO_STRING, tmp, 2);
tmp := BYTE_TO_STRING(DWORD_TO_BYTE(SHR(IP4,16)));
IP4_TO_STRING := INSERT(IP4_TO_STRING, tmp, 1);
tmp := BYTE_TO_STRING(DWORD_TO_BYTE(SHR(IP4,24)));
IP4_TO_STRING := CONCAT(tmp, IP4_TO_STRING);



(* revision history
hm	22. apr 2008	rev 1.0
	original version

hm	10. mar. 2009	rev 1.1
	improved code
*)
          
END_FUNCTION

FUNCTION IS_IP4 : BOOL
  VAR_INPUT
    str : STRING;
  END_VAR

            IS_IP4 := OSCAT_BASIC.COUNT_CHAR(str, 46) = 3;


(* revision history
hm	1. mar. 2008	rev 1.0
	original version

hm	10. mar. 2009	rev 1.1
	new code

*)
          
END_FUNCTION

FUNCTION IS_URLCHR : BOOL
  VAR_INPUT
    IN : BYTE;
  END_VAR

            IS_URLCHR := ((IN > 47) AND (IN < 58)) OR ((IN > 64) AND (IN < 91)) OR ((IN > 96) AND (IN < 123)) OR (in = 126) OR (in = 95) OR (in =45) OR (in =46);


(* revision history
hm		27. apr. 2008	rev 1.0
	original version

*)
          
END_FUNCTION

FUNCTION MD5_AUX : DWORD
  VAR_INPUT
    N : INT;
    A : DWORD;
    B : DWORD;
    C : DWORD;
    D : DWORD;
    X : DWORD;
    U : INT;
    T : DWORD;
  END_VAR
  VAR
    w : DWORD;
  END_VAR

            CASE N OF
	1: w := (B AND C) OR (NOT(B) AND D);
	2: w := (B AND D) OR (C AND NOT D);
	3: w := (B XOR C XOR D);
	4: w := (C XOR (B OR  NOT(D)));
END_CASE

MD5_AUX := B + ROL(A + w + X + T,U);

(* revision history

ks	6. dec. 2009 rev 1.0
	original version

*)
          
END_FUNCTION

FUNCTION_BLOCK MD5_CRAM_AUTH
  VAR_IN_OUT
    RUN : BOOL;
    USERNAME : STRING(64);
    PASSWORD : STRING(64);
    B64_TS : STRING(64);  (* Base64 coded ServerTimeStamp *)
    AUTH_KEY : STRING(192);
  END_VAR
  VAR
    BASE64_DECODE_STR : BASE64_DECODE_STR;
    BASE64_ENCODE_STR : BASE64_ENCODE_STR;
    MD5_STREAM : MD5_STREAM;
    step : INT;
    md5_mode : INT;
    buf : ARRAY[0..63] OF BYTE;
    md5 : ARRAY[0..15] OF BYTE;
    md5_first : ARRAY[0..15] OF BYTE;
    md5_str1 : STRING(64);
    md5_str2 : STRING(64);
    size : UDINT;
    n1 : INT;
    n2 : INT;
    pos : UDINT;
    b64d_run : BOOL;
    b64d_done : BOOL;
    b64e_run : BOOL;
    b64e_done : BOOL;
    str_192 : STRING(192);
    str_144 : STRING(144);
    xpad : BYTE;
    pt : POINTER TO BYTE;
  END_VAR

            CASE step OF

0:	IF RUN THEN
		step := 5;
		str_192 := B64_TS;
		b64d_run := TRUE;
	END_IF;

5: IF B64D_DONE THEN (* IPAD Zyklus *)
		b64d_run := FALSE;
		xpad := 16#36;
		md5_str1 := PASSWORD;
		md5_str2 := str_144;
		size := 64 + LEN(md5_str2);
		md5_mode := 1;
		step := 10;
	END_IF;

10: IF md5_mode = 3 THEN (* OPAD Zyklus *)
		md5_first := md5; (* md5 array vom IPAD sichern *)
		xpad := 16#5C;
		size := 64 + 16;
		md5_mode := 1;
		step := 20;
	END_IF;

20: IF md5_mode = 3 THEN
		md5_mode := 0;
		str_144 := CONCAT(USERNAME , ' ');
		str_144 := CONCAT(str_144 , MD5_TO_STRH(md5));
		b64e_run := TRUE;
		step := 30;
	END_IF;

30: IF B64E_DONE THEN
		AUTH_KEY := str_192;
		b64e_run := FALSE;
		RUN := FALSE;
		step := 0; (* alles beendet !! *)
	END_IF;

END_CASE;

(* ----------- md5 -------------- *)
CASE md5_mode OF

1:	n2 := LEN(md5_str1) - 1;
	pt := ADR(md5_str1);
	FOR n1 := 0 TO n2 DO (* string in buf kopieren *)
		buf[n1] := pt^ XOR xpad;
		pt := pt + 1;
	END_FOR;
	FOR n1 := n2 + 1 TO 63 DO (* mit ipad füllen *)
		buf[n1] := xpad;
	END_FOR;

2:	(* Data copy and Calc *)
	IF size > 0 AND pos >= 64 THEN
		IF step = 20 THEN
			FOR n1 := 0 TO 15 DO
				buf[n1] := md5_first[n1];
			END_FOR;
		ELSE
			n2 := LEN(md5_str2) - 1;
			pt := ADR(md5_str2);
			FOR n1 := 0 TO n2 DO (* string in buf kopieren *)
				buf[n1] := pt^;
				pt := pt + 1;
			END_FOR;
		END_IF;
	END_IF;

END_CASE;

IF md5_mode > 0 THEN
	MD5_STREAM(SIZE:=size, MODE:=md5_mode, BUF:=buf, MD5:=md5, POS=>pos);
END_IF;

BASE64_DECODE_STR(RUN:=b64d_run, STR1:=str_192, STR2:=str_144, DONE=>b64d_done);
BASE64_ENCODE_STR(RUN:=b64e_run, STR1:=str_144, STR2:=str_192, DONE=>b64e_done);

(* revision history

hm		10. mai. 2010	rev 1.0
	original version
*)
          
END_FUNCTION_BLOCK

FUNCTION_BLOCK MD5_STR
  VAR_INPUT
    RUN : BOOL;
  END_VAR
  VAR_OUTPUT
    DONE : BOOL;
  END_VAR
  VAR_IN_OUT
    STR : STRING(OSCAT_BASIC.STRING_LENGTH);
    MD5 : ARRAY[0..15] OF BYTE;
  END_VAR
  VAR
    run_last : BOOL;
    MD5_STREAM : MD5_STREAM;
    buf : ARRAY[0..63] OF BYTE;
    mode : INT;
    size : UDINT;
    pos : UDINT;
  END_VAR

            CASE mode OF
0:	(* Wait für Start *)
	IF RUN AND NOT run_last THEN
		DONE := FALSE;
		mode := 1; (* Initialisierung *)
		size := LEN(STR);
	END_IF;

2:	(* Data copy and Calc *)
	IF size > 0 THEN
		OSCAT_BASIC._STRING_TO_BUFFER(STR:=MID(STR, UDINT_TO_INT(SIZE), UDINT_TO_INT(POS) + 1), POS:=0, PT:=ADR(buf), SIZE:=SIZEOF(buf));
	END_IF;

3:	DONE := TRUE;
	mode := 0; (* Stop *)

END_CASE;

IF mode > 0 THEN
	MD5_STREAM(SIZE:=size, MODE:=mode, BUF:=buf, MD5:=MD5, POS=>pos);
END_IF;

run_last := RUN;

(* revision history

ks	6. dec. 2009 rev 1.0
	original version

*)
          
END_FUNCTION_BLOCK

FUNCTION_BLOCK MD5_STREAM
  VAR_IN_OUT
    MODE : INT;
    BUF : ARRAY[0..63] OF BYTE;
    MD5 : ARRAY[0..15] OF BYTE;
    SIZE : UDINT;
  END_VAR
  VAR_OUTPUT
    POS : UDINT;
  END_VAR
  VAR
    hash : ARRAY[0..3] OF DWORD;
    a : DWORD;
    b : DWORD;
    c : DWORD;
    d : DWORD;
    end : UDINT;
    block : UDINT;
    x : ARRAY[0..15] OF DWORD;
    n : INT;
    n1 : INT;
    z : INT;
    pad_1 : BOOL;
  END_VAR

            CASE MODE OF

1:	(* Initialisierung der Hash-Werte *)
	hash[0] := DWORD#16#67452301;
	hash[1] := DWORD#16#EFCDAB89;
	hash[2] := DWORD#16#98BADCFE;
	hash[3] := DWORD#16#10325476;

	block := SHR(SIZE,6) + BOOL_TO_UDINT((UDINT_TO_BYTE(SIZE) AND 16#3F) > 55);
	pad_1 := FALSE;
	POS := 0;
	End := SIZE;
	SIZE := MIN(64,End);
	MODE := 2;

2:	(* Fuell-Bytes anhängen *)
	FOR n := UDINT_TO_INT(SIZE) TO 63 DO
		BUF[n] := 0;
	END_FOR;

	IF SIZE < 64 AND NOT pad_1 THEN
		BUF[SIZE] := 2#1000_0000;
		pad_1 := TRUE;
	END_IF;

	POS := POS + SIZE;
	SIZE := MIN(64,End - POS);

	n := 0;	(* Byte-Array in DWORD-Array umkopieren *)
	FOR n1 := 0 TO 15 DO
		x[n1] := OSCAT_BASIC.DWORD_OF_BYTE(BUF[n+3],BUF[n+2],BUF[n+1],BUF[n]); (* Little Endian Format *)
		n := n + 4;
	END_FOR;

	IF block = 0 THEN (* am Ende des letzten Blocks die Datenlänge eintragen *)
		x[14] := SHL(UDINT_TO_DWORD(End),3); (* Anzahl Datenbits im Little-Endian Format eintragen *)
		MODE := 3;
	ELSE
		block := block - 1;
	END_IF;

	a := hash[0];
	b := hash[1];
	c := hash[2];
	d := hash[3];

	a := MD5_AUX(1, a, b, c, d, X[00], 07, 16#D76AA478); (* 01 *)
	d := MD5_AUX(1, d, a, b, c, X[01], 12, 16#E8C7B756); (* 02 *)
	c := MD5_AUX(1, c, d, a, b, X[02], 17, 16#242070DB); (* 03 *)
	b := MD5_AUX(1, b, c, d, a, X[03], 22, 16#C1BDCEEE); (* 04 *)
	a := MD5_AUX(1, a, b, c, d, X[04], 07, 16#F57C0FAF); (* 05 *)
	d := MD5_AUX(1, d, a, b, c, X[05], 12, 16#4787C62A); (* 06 *)
	c := MD5_AUX(1, c, d, a, b, X[06], 17, 16#A8304613); (* 07 *)
	b := MD5_AUX(1, b, c, d, a, X[07], 22, 16#FD469501); (* 08 *)
	a := MD5_AUX(1, a, b, c, d, X[08], 07, 16#698098D8); (* 09 *)
	d := MD5_AUX(1, d, a, b, c, X[09], 12, 16#8B44F7AF); (* 10 *)
	c := MD5_AUX(1, c, d, a, b, X[10], 17, 16#FFFF5BB1); (* 11 *)
	b := MD5_AUX(1, b, c, d, a, X[11], 22, 16#895CD7BE); (* 12 *)
	a := MD5_AUX(1, a, b, c, d, X[12], 07, 16#6B901122); (* 13 *)
	d := MD5_AUX(1, d, a, b, c, X[13], 12, 16#FD987193); (* 14 *)
	c := MD5_AUX(1, c, d, a, b, X[14], 17, 16#A679438E); (* 15 *)
	b := MD5_AUX(1, b, c, d, a, X[15], 22, 16#49B40821); (* 16 *)

	a := MD5_AUX(2, a, b, c, d, X[01], 05, 16#F61E2562); (* 17 *)
	d := MD5_AUX(2, d, a, b, c, X[06], 09, 16#C040B340); (* 18 *)
	c := MD5_AUX(2, c, d, a, b, X[11], 14, 16#265E5A51); (* 19 *)
	b := MD5_AUX(2, b, c, d, a, X[00], 20, 16#E9B6C7AA); (* 20 *)
	a := MD5_AUX(2, a, b, c, d, X[05], 05, 16#D62F105D); (* 21 *)
	d := MD5_AUX(2, d, a, b, c, X[10], 09, 16#02441453); (* 22 *)
	c := MD5_AUX(2, c, d, a, b, X[15], 14, 16#D8A1E681); (* 23 *)
	b := MD5_AUX(2, b, c, d, a, X[04], 20, 16#E7D3FBC8); (* 24 *)
	a := MD5_AUX(2, a, b, c, d, X[09], 05, 16#21E1CDE6); (* 25 *)
	d := MD5_AUX(2, d, a, b, c, X[14], 09, 16#C33707D6); (* 26 *)
	c := MD5_AUX(2, c, d, a, b, X[03], 14, 16#F4D50D87); (* 27 *)
	b := MD5_AUX(2, b, c, d, a, X[08], 20, 16#455A14ED); (* 28 *)
	a := MD5_AUX(2, a, b, c, d, X[13], 05, 16#A9E3E905); (* 29 *)
	d := MD5_AUX(2, d, a, b, c, X[02], 09, 16#FCEFA3F8); (* 30 *)
	c := MD5_AUX(2, c, d, a, b, X[07], 14, 16#676F02D9); (* 31 *)
	b := MD5_AUX(2, b, c, d, a, X[12], 20, 16#8D2A4C8A); (* 32 *)

	a := MD5_AUX(3, a, b, c, d, X[05], 04, 16#FFFA3942); (* 33 *)
	d := MD5_AUX(3, d, a, b, c, X[08], 11, 16#8771F681); (* 34 *)
	c := MD5_AUX(3, c, d, a, b, X[11], 16, 16#6D9D6122); (* 35 *)
	b := MD5_AUX(3, b, c, d, a, X[14], 23, 16#FDE5380C); (* 36 *)
	a := MD5_AUX(3, a, b, c, d, X[01], 04, 16#A4BEEA44); (* 37 *)
	d := MD5_AUX(3, d, a, b, c, X[04], 11, 16#4BDECFA9); (* 38 *)
	c := MD5_AUX(3, c, d, a, b, X[07], 16, 16#F6BB4B60); (* 39 *)
	b := MD5_AUX(3, b, c, d, a, X[10], 23, 16#BEBFBC70); (* 40 *)
	a := MD5_AUX(3, a, b, c, d, X[13], 04, 16#289B7EC6); (* 41 *)
	d := MD5_AUX(3, d, a, b, c, X[00], 11, 16#EAA127FA); (* 42 *)
	c := MD5_AUX(3, c, d, a, b, X[03], 16, 16#D4EF3085); (* 43 *)
	b := MD5_AUX(3, b, c, d, a, X[06], 23, 16#04881D05); (* 44 *)
	a := MD5_AUX(3, a, b, c, d, X[09], 04, 16#D9D4D039); (* 45 *)
	d := MD5_AUX(3, d, a, b, c, X[12], 11, 16#E6DB99E5); (* 46 *)
	c := MD5_AUX(3, c, d, a, b, X[15], 16, 16#1FA27CF8); (* 47 *)
	b := MD5_AUX(3, b, c, d, a, X[02], 23, 16#C4AC5665); (* 48 *)

	a := MD5_AUX(4, a, b, c, d, X[00], 06, 16#F4292244); (* 49 *)
	d := MD5_AUX(4, d, a, b, c, X[07], 10, 16#432AFF97); (* 50 *)
	c := MD5_AUX(4, c, d, a, b, X[14], 15, 16#AB9423A7); (* 51 *)
	b := MD5_AUX(4, b, c, d, a, X[05], 21, 16#FC93A039); (* 52 *)
	a := MD5_AUX(4, a, b, c, d, X[12], 06, 16#655B59C3); (* 53 *)
	d := MD5_AUX(4, d, a, b, c, X[03], 10, 16#8F0CCC92); (* 54 *)
	c := MD5_AUX(4, c, d, a, b, X[10], 15, 16#FFEFF47D); (* 55 *)
	b := MD5_AUX(4, b, c, d, a, X[01], 21, 16#85845DD1); (* 56 *)
	a := MD5_AUX(4, a, b, c, d, X[08], 06, 16#6FA87E4F); (* 57 *)
	d := MD5_AUX(4, d, a, b, c, X[15], 10, 16#FE2CE6E0); (* 58 *)
	c := MD5_AUX(4, c, d, a, b, X[06], 15, 16#A3014314); (* 59 *)
	b := MD5_AUX(4, b, c, d, a, X[13], 21, 16#4E0811A1); (* 60 *)
	a := MD5_AUX(4, a, b, c, d, X[04], 06, 16#F7537E82); (* 61 *)
	d := MD5_AUX(4, d, a, b, c, X[11], 10, 16#BD3AF235); (* 62 *)
	c := MD5_AUX(4, c, d, a, b, X[02], 15, 16#2AD7D2BB); (* 63 *)
	b := MD5_AUX(4, b, c, d, a, X[09], 21, 16#EB86D391); (* 64 *)

	hash[0] := hash[0] + a;
	hash[1] := hash[1] + b;
	hash[2] := hash[2] + c;
	hash[3] := hash[3] + d;

END_CASE;

IF MODE = 3 THEN
	z := 0;
	FOR n := 0 TO 3 DO (* von Little-Endian auf Big-Endian format konvertieren und DWORD auf BYTE-Array *)
		FOR n1 := 0 TO 3 DO
			MD5[z] := DWORD_TO_BYTE(hash[n]);
			hash[n] := ROR(hash[n],8);
			z := z + 1;
		END_FOR;
	END_FOR;
END_IF;

(* revision history

ks	6. dec. 2009 rev 1.0
	original version

*)
          
END_FUNCTION_BLOCK

FUNCTION MD5_TO_STRH : STRING(32)
  VAR_INPUT
    MD5 : ARRAY[0..15] OF BYTE;
  END_VAR
  VAR
    i : INT;
    tmp : BYTE;
    pt : POINTER TO BYTE;
  END_VAR

            pt := ADR(MD5_TO_STRH); (* read output adress to pointer *)

FOR i := 0 TO 15 DO; (* write the 8 hex characters backwards *)
	tmp := SHR(MD5[i],4);
	PT^ := tmp + SEL(tmp <= 9,87,48);
	pt := pt + 1; (* decrement the pointer *)
	tmp := MD5[i] AND 2#1111;
	PT^ := tmp + SEL(tmp <= 9,87,48);
	pt := pt + 1; (* decrement the pointer *)
END_FOR;
pt^:= 0; (* write the closing byte for the string *)

(* revision history

ks	6. dec. 2009 rev 1.0
	original version

*)
          
END_FUNCTION

FUNCTION_BLOCK RC4_CRYPT_STREAM
  VAR_IN_OUT
    MODE : INT;
    KEY : STRING(40);
    BUF : ARRAY[0..63] OF BYTE;
    SIZE : UDINT;
  END_VAR
  VAR_OUTPUT
    POS : UDINT;
  END_VAR
  VAR
    sbox : ARRAY[0..255] OF BYTE;
    skey : ARRAY[0..255] OF BYTE;
    a : INT;
    b : INT;
    c : INT;
    d : USINT;
    e : USINT;
    end : UDINT;
    v : BYTE;
  END_VAR

            CASE MODE OF

1:	(* Initialisierung *)
	b := LEN(KEY) - 1;
	IF b < 0 OR SIZE < 1 THEN
		MODE := 3;
		RETURN;
	END_IF;

	FOR a := 0 TO b DO
		skey[a] := OSCAT_BASIC.CODE(KEY, a + 1);
		sbox[a] := INT_TO_BYTE(a);
	END_FOR;

	c := 0;
	FOR a := b + 1 TO 255 DO
		skey[a] := skey[c];
		sbox[a] := INT_TO_BYTE(a);
		c := c + 1;
		IF c > b THEN c := 0; END_IF;
	END_FOR;

	d := 0;
	FOR a := 0 TO 255 DO
		d := d + sbox[a] + skey[a];
		v := sbox[a];
		sbox[a] := sbox[d];
		sbox[d] := v;
	END_FOR;

	POS := 0;
	end := SIZE;
	SIZE := MIN(64,end);
	d := 0;
	e := 0;
	MODE := 2;

2:	(* Daten ver/entschlüsseln *)

	b := UDINT_TO_INT(SIZE) - 1;
	FOR a := 0 TO b DO
		d := d + 1;
		e := e + sbox[d];
		v := sbox[d];
		sbox[d] := sbox[e];
		sbox[e] := v;
		v := sbox[d] + sbox[e];
		BUF[a] :=BUF[a] XOR sbox[v];
	END_FOR;

	POS := POS + SIZE;
	SIZE := MIN(64,end - POS);

	IF SIZE = 0 THEN
		MODE := 3;
	END_IF;
END_CASE;

(* revision history

ks	9. Jan. 2010 rev 1.0
	original version

*)
          
END_FUNCTION_BLOCK

FUNCTION_BLOCK SHA1_STR
  VAR_INPUT
    RUN : BOOL;
  END_VAR
  VAR_OUTPUT
    DONE : BOOL;
  END_VAR
  VAR_IN_OUT
    STR : STRING(OSCAT_BASIC.STRING_LENGTH);
    SHA1 : ARRAY[0..19] OF BYTE;
  END_VAR
  VAR
    run_last : BOOL;
    SHA1_STREAM : SHA1_STREAM;
    buf : ARRAY[0..63] OF BYTE;
    mode : INT;
    size : UDINT;
    pos : UDINT;
  END_VAR

            CASE mode OF
0:	(* Wait für Start *)
	IF RUN AND NOT run_last THEN
		DONE := FALSE;
		mode := 1; (* Initialisierung *)
		size := LEN(STR);
	END_IF;

2:	(* Data copy and Calc *)
	IF size > 0 THEN
		OSCAT_BASIC._STRING_TO_BUFFER(STR:=MID(STR, UDINT_TO_INT(SIZE), UDINT_TO_INT(POS) + 1), POS:=0, PT:=ADR(buf), SIZE:=SIZEOF(buf));
	END_IF;

3:	DONE := TRUE;
	mode := 0; (* Stop *)

END_CASE;

IF mode > 0 THEN
	SHA1_STREAM(SIZE:=size, MODE:=mode, BUF:=buf, SHA1:=SHA1, POS=>pos);
END_IF;

run_last := RUN;

(* revision history

ks	6. dec. 2009 rev 1.0
	original version

*)
          
END_FUNCTION_BLOCK

FUNCTION_BLOCK SHA1_STREAM
  VAR_IN_OUT
    MODE : INT;
    BUF : ARRAY[0..63] OF BYTE;
    SHA1 : ARRAY[0..19] OF BYTE;
    SIZE : UDINT;
  END_VAR
  VAR_OUTPUT
    POS : UDINT;
  END_VAR
  VAR
    hash : ARRAY[0..4] OF DWORD;
    end : UDINT;
    block : UDINT;
    pad_1 : BOOL;
    w : ARRAY[0..79] OF DWORD;
    n : INT;
    n1 : INT;
    a : DWORD;
    b : DWORD;
    c : DWORD;
    d : DWORD;
    e : DWORD;
    f : DWORD;
    k : DWORD;
    x : DWORD;
    z : INT;
  END_VAR

            CASE MODE OF

1:	(* Initialisierung der Hash-Werte *)
	hash[0] := DWORD#16#67452301;
	hash[1] := DWORD#16#EFCDAB89;
	hash[2] := DWORD#16#98BADCFE;
	hash[3] := DWORD#16#10325476;
	hash[4] := DWORD#16#C3D2E1F0;

	(* Buffer initialisieren *)
	FOR n := 16 TO 79 DO
   		w[n] := DWORD#0;
	END_FOR;

	block := SHR(SIZE,6) + BOOL_TO_UDINT((UDINT_TO_BYTE(SIZE) AND 16#3F) > 55);	(* benötigte Blocks errechnen *)

	pad_1 := FALSE;
	POS := 0;
	End := SIZE;
	SIZE := MIN(64,End);
	MODE := 2;

2:	FOR n := UDINT_TO_INT(SIZE) TO 63 DO (* Fuell-Bytes anhängen *)
		BUF[n] := 0;
	END_FOR;

	IF SIZE < 64 AND NOT pad_1 THEN
		BUF[SIZE] := 2#1000_0000;
		pad_1 := TRUE;
	END_IF;

	POS := POS + SIZE;
	SIZE := MIN(64,End - POS);

	n := 0;	(* Byte-Array in DWORD-Array umkopieren *)
	FOR n1 := 0 TO 15 DO
		w[n1] := OSCAT_BASIC.DWORD_OF_BYTE(BUF[n],BUF[n+1],BUF[n+2],BUF[n+3]);
		n := n + 4;
	END_FOR;

	IF block = 0 THEN (* am Ende des letzten Blocks die Datenlänge eintragen *)
		w[15] := SHL(UDINT_TO_DWORD(End),3); (* Anzahl Datenbits eintragen *)
		MODE := 3;
	ELSE
		block := block - 1;
	END_IF;

	FOR n := 16 TO 79 DO (* erweitern der 16 32-bit-Worte auf 80 32-bit-Worte *)
		w[n] := ROL(w[n-3] XOR w[n-8] XOR w[n-14] XOR w[n-16],1);
	END_FOR;

	a := hash[0];
	b := hash[1];
	c := hash[2];
	d := hash[3];
	e := hash[4];

	FOR n := 0 TO 79 DO
		IF n <= 19 THEN
			f := (b AND c) OR (NOT(b) AND d);
			k := DWORD#16#5A827999;
		ELSIF n <= 39 THEN
			f := b XOR c XOR d;
			k := DWORD#16#6ED9EBA1;
		ELSIF n <= 59 THEN
			f := (b AND c) OR (b AND d) OR (c AND d);
			k := DWORD#16#8F1BBCDC;
		ELSE
			f := b XOR c XOR d;
			k := DWORD#16#CA62C1D6;
		END_IF;

		x := ROL(a,5) + f + e + k + w[n];
		e := d;
		d := c;
		c := ROL(b,30);
		b := a;
		a := x;
	END_FOR;

	(* aktuelle Hash-Werte zum letzten Wert addieren *)
	hash[0] := hash[0] + a;
	hash[1] := hash[1] + b;
	hash[2] := hash[2] + c;
	hash[3] := hash[3] + d;
	hash[4] := hash[4] + e;

END_CASE;

IF MODE = 3 THEN
	z := 0;
	FOR n := 0 TO 4 DO (* konvertiere DWORD auf BYTE-Array *)
		FOR n1 := 0 TO 3 DO
			hash[n] := ROL(hash[n],8);
			SHA1[z] := DWORD_TO_BYTE(hash[n]);
			z := z + 1;
		END_FOR;
	END_FOR;
END_IF;

(* revision history

ks	6. dec. 2009 rev 1.0
	original version

*)
          
END_FUNCTION_BLOCK

FUNCTION SHA1_TO_STRH : STRING(40)
  VAR_INPUT
    SHA1 : ARRAY[0..19] OF BYTE;
  END_VAR
  VAR
    i : INT;
    tmp : BYTE;
    pt : POINTER TO BYTE;
  END_VAR

            pt := ADR(SHA1_TO_STRH); (* read output adress to pointer *)

FOR i := 0 TO 19 DO; (* write the 10 hex characters backwards *)
	tmp := SHR(SHA1[i],4);
	PT^ := tmp + SEL(tmp <= 9,87,48);
	pt := pt + 1; (* decrement the pointer *)
	tmp := SHA1[i] AND 2#1111;
	PT^ := tmp + SEL(tmp <= 9,87,48);
	pt := pt + 1; (* decrement the pointer *)
END_FOR;
pt^:= 0; (* write the closing byte for the string *)

(* revision history

ks	6. dec. 2009 rev 1.0
	original version

ks	3. dec. 2011 rev 1.1
	incorrect string size
*)
          
END_FUNCTION

FUNCTION STRING_TO_URL : URL
  VAR_INPUT
    STR : STRING(OSCAT_BASIC.STRING_LENGTH);
    DEFAULT_PROTOCOL : STRING(10);
    DEFAULT_PATH : STRING(80);
  END_VAR
  VAR
    pos : INT;
    pos2 : INT;
    x : STRING(OSCAT_BASIC.STRING_LENGTH);
  END_VAR

            (*

http://hans:geheim@www.example.org:80/demo/example.cgi?land=de&stadt=aa#abschnitt1
|       |      |         |         |   |                   |               |
|       |      |         Host      |   Pfad                Query           Anker
|       |      Passwort            Port
|       Benutzer
Protokoll

*)

(* check if string is empty and return empty url *)
IF STR = '' THEN RETURN; END_IF;

(* extract the protocol *)
(* first we check if the optional protocol is specified ending with a :// *)
pos := FIND(STR, '://');
IF pos > 0 THEN
	(* store protocol and restore the rest of url in temp *)
	STRING_TO_URL.PROTOCOL := LEFT(STR, pos - 1);
	x := RIGHT(STR, LEN(STR) - pos - 2);
ELSE
	x := STR;
	STRING_TO_URL.PROTOCOL := DEFAULT_PROTOCOL;
END_IF;

(* extract user and password if present ending with a @ *)
pos := OSCAT_BASIC.FINDB(STR1:=x,STR2:='@'); (* Find last @ *)

IF pos > 0 THEN
	(* extract user *)
	pos2 := FIND(x,':')+1;
	IF pos2 > 1 AND pos2 <= pos THEN
		STRING_TO_URL.USER := LEFT(x,pos2 - 2);
		STRING_TO_URL.PASSWORD := MID(x, pos - pos2, pos2);
	ELSE
		STRING_TO_URL.USER := LEFT(x, pos - 2);
		STRING_TO_URL.PASSWORD := '';
	END_IF;
	x := RIGHT(x, LEN(x) - pos);
ELSE
	STRING_TO_URL.USER := '';
	STRING_TO_URL.PASSWORD := '';
END_IF;

(* extract anchor *)
pos := FIND(x, '#');
IF pos > 0 THEN
	STRING_TO_URL.ANCHOR := RIGHT(x, LEN(x) - pos);
	x := LEFT(x, pos - 1);
ELSE
	STRING_TO_URL.ANCHOR := '';
END_IF;

(* extract query  *)
pos := FIND(x, '?');
IF pos > 0 THEN
	STRING_TO_URL.QUERY := RIGHT(x, LEN(x) - pos);
	x := LEFT(x, pos - 1);
ELSE
	STRING_TO_URL.QUERY := '';
END_IF;

(* extract path  *)
pos := FIND(x, '/');
IF pos > 0 THEN
	STRING_TO_URL.PATH := RIGHT(x, LEN(x) - pos + 1);
	x := LEFT(x, pos - 1);
ELSE
	STRING_TO_URL.PATH := DEFAULT_PATH;
END_IF;

(* extract port and leave domain *)
pos := FIND(x, ':');
IF pos > 0 THEN
	STRING_TO_URL.PORT := STRING_TO_WORD(RIGHT(x, LEN(x) - pos));
	STRING_TO_URL.DOMAIN := LEFT(x, pos - 1);
ELSE
	STRING_TO_URL.PORT := 0;
	STRING_TO_URL.DOMAIN := x;
END_IF;

(* revision history
hm		18. apr 2008	rev 1.0
	original version

ks		20. dec. 2010	rev 1.1
	stringlength 250 , var x

ks		27. oct. 2012	rev 1.2
	var_temp zu var geändert

ks		04. mar. 2016	rev 1.3
	@ zeichen wird nun von rechts nach links gesucht
	ermöglicht username und password mit @ zeichen
*)
          
END_FUNCTION

FUNCTION URL_DECODE : STRING(OSCAT_BASIC.STRING_LENGTH)
  VAR_INPUT
    IN : STRING(OSCAT_BASIC.STRING_LENGTH);
  END_VAR
  VAR
    pos : INT;
    seq : STRING(3);
    new : STRING(1);
  END_VAR

            URL_DECODE := IN;
pos := FIND(URL_DECODE,'%');
WHILE pos > 0 DO
	seq := MID(URL_DECODE,2,pos + 1);
	new := OSCAT_BASIC.CHR_TO_STRING(DWORD_TO_BYTE(OSCAT_BASIC.HEX_TO_DWORD(seq)));
	URL_DECODE := REPLACE(URL_DECODE, new, 3, pos);
	pos := FIND(URL_DECODE,'%');
END_WHILE;


(* revision history
hm	27. apr. 2008	rev 1.0
	original version

hm	17. dec. 2008	rev 1.1
	changes name of function chr to chr_to_string

ks	10. mai. 2008	rev 1.2
	stringlength 250
*)
          
END_FUNCTION

FUNCTION URL_ENCODE : STRING(OSCAT_BASIC.STRING_LENGTH)
  VAR_INPUT
    IN : STRING(OSCAT_BASIC.STRING_LENGTH);
  END_VAR
  VAR
    pt_in : POINTER TO ARRAY[1..255] OF BYTE;
    pt_out : POINTER TO ARRAY[1..256] OF BYTE;
    pos_in : INT;
    pos_out : INT;
    stop : INT;
    tb : BYTE;
  END_VAR

            pt_in  := ADR(in);
pt_out := ADR(URL_ENCODE);

(* scan the input string and convert unallowed characters *)
pos_in := 1;
stop := LEN(in);
FOR pos_out := 1 TO 250 DO
	IF pos_in > stop THEN
		EXIT;
	ELSIF IS_URLCHR(pt_in^[pos_in]) THEN
		pt_out^[pos_out] := pt_in^[pos_in];
		(* increment in by 1 *)
		pos_in := pos_in + 1;
	ELSE
		(* cannot fit 3 digits, exit *)
		IF pos_out > 248 THEN EXIT; END_IF;
		(* invalid character that needs to be converted *)
		pt_out^[pos_out] := 37;    (* start with % sign *)
		pos_out := pos_out + 1;
		(* need to add the two hex digits *)
		tb := SHR(pt_in^[pos_in],4);
		IF tb > 9 THEN
			pt_out^[pos_out] := tb + 55;
		ELSE
			pt_out^[pos_out] := tb + 48;
		END_IF;
		pos_out := pos_out + 1;
		tb := pt_in^[pos_in] AND 16#0F;
		IF tb > 9 THEN
			pt_out^[pos_out] := tb + 55;
		ELSE
			pt_out^[pos_out] := tb + 48;
		END_IF;
		(* increment in and out because out has to move 3 digits *)
		pos_in := pos_in + 1;
	END_IF;
END_FOR;

(* terminate the output string *)
pt_out^[pos_out] := 0;

(* revision history
hm	27. apr. 2008	rev 1.0
	original version

ks	10. mai. 2008	rev 1.1
	stringlength 250

*)
          
END_FUNCTION

FUNCTION URL_TO_STRING : STRING(OSCAT_BASIC.STRING_LENGTH)
  VAR_INPUT
    IN : URL;
  END_VAR

            (*

http://hans:geheim@www.example.org:80/demo/example.cgi?land=de&stadt=aa#abschnitt1
|         |         |                  |                                |   |                                    |                                    |
|         |         |                 Host                         |   Pfad                            Query                           Anker
|         |         Passwort                                  Port
|        Benutzer
Protokoll

*)

(* attach protocol *)
IF IN.PROTOCOL <> '' THEN URL_TO_STRING := CONCAT(IN.PROTOCOL,'://'); END_IF;

(* attach user and password *)
IF IN.USER <> '' THEN
	URL_TO_STRING := CONCAT(URL_TO_STRING, IN.USER);
	IF IN.PASSWORD <> '' THEN
		URL_TO_STRING := CONCAT(URL_TO_STRING, ':');
		URL_TO_STRING := CONCAT(URL_TO_STRING, IN.PASSWORD);
	END_IF;
	URL_TO_STRING := CONCAT(URL_TO_STRING, '@');
END_IF;

(* attach domain *)
URL_TO_STRING := CONCAT(URL_TO_STRING, IN.DOMAIN);

(* attach Port *)
IF IN.PORT > 0 THEN
	URL_TO_STRING := CONCAT(URL_TO_STRING, ':');
	URL_TO_STRING := CONCAT(URL_TO_STRING, WORD_TO_STRING(IN.PORT));
END_IF;

(* attach path *)
URL_TO_STRING := CONCAT(URL_TO_STRING, IN.PATH);

(* attach query *)
IF IN.QUERY <> '' THEN
	URL_TO_STRING := CONCAT(URL_TO_STRING, '?');
	URL_TO_STRING := CONCAT(URL_TO_STRING, IN.QUERY);
END_IF;

(* attach anchor *)
IF IN.ANCHOR <> '' THEN
	URL_TO_STRING := CONCAT(URL_TO_STRING, '#');
	URL_TO_STRING := CONCAT(URL_TO_STRING, IN.ANCHOR);
END_IF;

(* revision history
hm	18. apr 2008	rev 1.0
	original version

ks	10. mai. 2008	rev 1.1
	stringlength 250
*)
          
END_FUNCTION

FUNCTION_BLOCK DLOG_BOOL
  VAR_IN_OUT
    X : DLOG_DATA;
  END_VAR
  VAR_INPUT
    STATE : BOOL;
    OFF : STRING;
    ON : STRING;
    COLUMN : STRING(40);
    DELTA : BOOL;
  END_VAR
  VAR
    UCB : UNI_CIRCULAR_BUFFER;
    id : WORD;
    last_delta : BOOL;
    state_last : BOOL;
  END_VAR

            CASE x.ADD_COM OF

01:	(* ADD INFO *)
	X.ID_MAX := X.ID_MAX + USINT#1;
	id := WORD#16#0601; (* Quelltype BOOL , Zieltype STRING *)
02:	(* ADD HEADER *)
	X.UCB.D_STRING := COLUMN;
	X.UCB.D_HEAD := id;
	X.UCB.D_MODE := 1;
	UCB(DATA:=X.UCB); (* Daten eintragen *)
03:	(* ADD DATA *)
	IF X.STORE_TYPE = BYTE#05 THEN (* MySQL-Modus *)
		X.UCB.D_STRING := SEL(state_last,'0','1');
	ELSE
		X.UCB.D_STRING := SEL(state_last,OFF,ON);
	END_IF;
	X.UCB.D_HEAD := id;

	X.UCB.D_MODE := 1;
	UCB(DATA:=X.UCB); (* Daten eintragen *)
	last_delta := STATE;
04:	(* ADD DATA REQ *)
	IF DELTA AND (STATE XOR last_delta) THEN
		X.ADD_DATA_REQ := TRUE;
		last_delta := STATE;
	END_IF;
END_CASE;
state_last := STATE;

(* revision history
ks	17. may. 2011	rev 1.0
	original version

ks	25. july.   2011	rev 1.1
	neue head information

ks	19. apr.   2012	rev 1.2
	code neu überarbeitet

*)
          
END_FUNCTION_BLOCK

FUNCTION_BLOCK DLOG_CRON_TAB
  VAR_INPUT
    ACTIVATE : BOOL;
    DTI : DT;
    SECOND : STRING(20);
    MINUTE : STRING(20);
    HOUR : STRING(20);
    DAY_OF_MONTH : STRING(20);
    DAY_OF_WEEK : STRING(20);
    MONTH : STRING(20);
  END_VAR
  VAR_OUTPUT
    Q : BOOL;
  END_VAR
  VAR
    CD : DLOG_CRON_DATA;
    activate_old : BOOL;
    datei : DATE;
    dti_last : DT;
    cnt1 : INT;
    cnt2 : INT;
    idx1 : INT;
    idx2 : INT;
    idx3 : INT;
    idx4 : INT;
    pos1 : INT;
    pos2 : INT;
    char_cnt : INT;
    trig_day : BOOL;
    trig_weekday : BOOL;
    str1 : STRING(OSCAT_BASIC.STRING_LENGTH);
    str2 : STRING(OSCAT_BASIC.STRING_LENGTH);
    str3 : STRING(OSCAT_BASIC.STRING_LENGTH);
    num_str1 : STRING(10);
  END_VAR

            IF ACTIVATE THEN
	IF NOT activate_old THEN
		CD.CE[0].VALUE_MIN := 0;	(* Sekunden *)
		CD.CE[0].VALUE_MAX := 59;
		CD.CE[1].VALUE_MIN := 0;	(* Minuten *)
		CD.CE[1].VALUE_MAX := 59;
		CD.CE[2].VALUE_MIN := 0;	(* Stunden *)
		CD.CE[2].VALUE_MAX := 59;
		CD.CE[3].VALUE_MIN := 1;	(* Tage *)
		CD.CE[3].VALUE_MAX := 31;
		CD.CE[4].VALUE_MIN := 1;	(* Wochentag *)
		CD.CE[4].VALUE_MAX := 7;
		CD.CE[5].VALUE_MIN := 1;	(* Monat *)
		CD.CE[5].VALUE_MAX := 12;

		FOR idx1 := 0 TO 5 DO
			idx3 := CD.CE[idx1].VALUE_MIN;
			idx4 := CD.CE[idx1].VALUE_MAx;
			FOR idx2 := idx3 TO idx4 DO
				CD.CE[idx1].ELEMENTS[idx2] := FALSE;
			END_FOR;
			CD.CE[idx1].ALL_SELECTED := FALSE;
		END_FOR;

		str1 := CONCAT(SECOND,'#');
		str1 := CONCAT(str1,MINUTE);
		str1 := CONCAT(str1,'#');
		str1 := CONCAT(str1,HOUR);
		str1 := CONCAT(str1,'#');
		str1 := CONCAT(str1,DAY_OF_MONTH);
		str1 := CONCAT(str1,'#');
		str1 := CONCAT(str1,DAY_OF_WEEK);
		str1 := CONCAT(str1,'#');
		str1 := CONCAT(str1,MONTH);

		FOR idx1 := 0 TO 5 DO
			str2 := ELEMENT_GET(BYTE#35, idx1, str1);
			IF LEN(str2) > 0 THEN
				cnt1 := ELEMENT_COUNT(BYTE#44, str2);	(* Trenzeichen ',' *)
			ELSE
				cnt1 := 1;
			END_IF;

			FOR idx2 := 0 TO cnt1 -1 DO
				str3 := ELEMENT_GET(BYTE#44, idx2, str2);
				IF FIND(str3, '*/') > 0 AND LEN(str3) <= 10 THEN
					pos1 := OSCAT_BASIC.DEC_TO_INT(str3);
					IF pos1 > 0 THEN
						idx3 := CD.CE[idx1].VALUE_MIN;
						idx4 := CD.CE[idx1].VALUE_MAX;
						WHILE idx3 <= idx4 DO
							CD.CE[idx1].ELEMENTS[idx3] := TRUE;
							idx3 := idx3 + pos1;
						END_WHILE;
					END_IF;

				ELSE
					IF FIND(str3, '*') > 0 OR LEN(str3) = 0 THEN
						pos1 := CD.CE[idx1].VALUE_MIN;
						pos2 := CD.CE[idx1].VALUE_MAX;
						CD.CE[idx1].ALL_SELECTED := TRUE;
					ELSE
						cnt2 := ELEMENT_COUNT(BYTE#45, str3);	(* Trenzeichen '-' *)
						char_cnt := LEN(str3);
						IF char_cnt >= 1 AND char_cnt <= 10 THEN
							num_str1 := ELEMENT_GET(BYTE#45, 0, str3);
							pos1 := OSCAT_BASIC.DEC_TO_INT(num_str1);
							pos2 := pos1;
							IF cnt2 = 2 THEN
								num_str1 := ELEMENT_GET(BYTE#45, 1, str3);
								pos2 := OSCAT_BASIC.DEC_TO_INT(num_str1);
							END_IF;
						END_IF;
					END_IF;

					IF pos1 >= CD.CE[idx1].VALUE_MIN AND pos2 <= CD.CE[idx1].VALUE_MAX THEN
						FOR idx3 := pos1 TO pos2 DO
							CD.CE[idx1].ELEMENTS[idx3] := TRUE;
						END_FOR;
					END_IF;
				END_IF;
			END_FOR;
		END_FOR;
	ELSIF DTI <> dti_last THEN
		CD.CE[0].VALUE := OSCAT_BASIC.SECOND_OF_DT(DTI); (* Sekunden *)
		CD.CE[1].VALUE := OSCAT_BASIC.MINUTE_OF_DT(DTI); (* Minuten *)
		CD.CE[2].VALUE := OSCAT_BASIC.HOUR_OF_DT(DTI); (* Stunden *)
		datei := DT_TO_DATE(DTI);
		CD.CE[3].VALUE := OSCAT_BASIC.DAY_OF_MONTH(datei); (* Tag *)
		CD.CE[4].VALUE := OSCAT_BASIC.DAY_OF_WEEK(datei); (* Wochentag *)
		CD.CE[5].VALUE := OSCAT_BASIC.MONTH_OF_DATE(datei); (*  Monat *)
		dti_last := DTI;

		idx2 := CD.CE[0].VALUE;	(* sekunden *)
		Q := CD.CE[0].ELEMENTS[idx2] = TRUE;
		idx2 := CD.CE[1].VALUE;	(* minuten *)
		Q := Q AND CD.CE[1].ELEMENTS[idx2] = TRUE;
		idx2 := CD.CE[2].VALUE;	(* stunden *)
		Q := Q AND CD.CE[2].ELEMENTS[idx2] = TRUE;
		idx2 := CD.CE[5].VALUE;	(* monat *)
		Q := Q AND CD.CE[5].ELEMENTS[idx2] = TRUE;

		(* auswertung Tag und Wochentag *)
		idx2 := CD.CE[3].VALUE;	(* Tag *)
		trig_day:= CD.CE[3].ELEMENTS[idx2] = TRUE;
		idx2 := CD.CE[4].VALUE;	(* Wochentag *)
		trig_weekday := CD.CE[4].ELEMENTS[idx2] = TRUE;

		IF CD.CE[3].ALL_SELECTED = FALSE AND CD.CE[4].ALL_SELECTED = TRUE THEN
			Q := Q AND trig_day; (* nur Tag auswerten *)
		ELSIF CD.CE[3].ALL_SELECTED = TRUE AND CD.CE[4].ALL_SELECTED = FALSE THEN
			Q := Q AND trig_weekday; (* nur Wochentag auswerten *)
		ELSIF CD.CE[3].ALL_SELECTED = FALSE AND CD.CE[4].ALL_SELECTED = FALSE THEN
			Q := Q AND (trig_weekday OR trig_day); (* Tag und Wochentag auswerten *)
		END_IF;
	END_IF;

END_IF;
activate_old := ACTIVATE;

(* revision history
ks	27. oct. 2011	rev 1.0
	original version
*)
          
END_FUNCTION_BLOCK

FUNCTION_BLOCK DLOG_DINT
  VAR_IN_OUT
    X : DLOG_DATA;
  END_VAR
  VAR_INPUT
    VALUE : DINT;
    COLUMN : STRING(40);
    DELTA : DINT;
  END_VAR
  VAR
    UCB : UNI_CIRCULAR_BUFFER;
    id : WORD;
    delta_last : DINT;
    value_last : DINT;
  END_VAR

            CASE x.ADD_COM OF

01:	(* ADD INFO *)
	X.ID_MAX := X.ID_MAX + USINT#1;
	id := WORD#16#0801; (* Quelltype DINT , Zieltype STRING *)
02:	(* ADD HEADER *)
	X.UCB.D_STRING := COLUMN;
	X.UCB.D_HEAD := id;
	X.UCB.D_MODE := 1;
	UCB(DATA:=X.UCB); (* Daten eintragen *)
03:	(* ADD DATA *)
	X.UCB.D_STRING := DINT_TO_STRING(value_last);
	X.UCB.D_HEAD := id;
	X.UCB.D_MODE := 1;
	UCB(DATA:=X.UCB); (* Daten eintragen *)
	delta_last := value_last;
04:	(* ADD DATA REQ *)
	IF DELTA <> DINT#0 THEN
		IF VALUE <= (delta_last - DELTA) OR VALUE >= (delta_last + DELTA) THEN
			X.ADD_DATA_REQ := TRUE;
			delta_last := VALUE;
		END_IF;
	END_IF;
END_CASE;
value_last := VALUE;

(* revision history
ks	01. jan. 2011	rev 1.0
	original version

ks	17. may. 2011	rev 1.1
	DELTA Funktion integriert

ks	25. july.   2011	rev 1.2
	neue head information

ks	19. apr.   2012	rev 1.2
	code neu überarbeitet
*)
          
END_FUNCTION_BLOCK

FUNCTION_BLOCK DLOG_DT
  VAR_IN_OUT
    X : DLOG_DATA;
  END_VAR
  VAR_INPUT
    FMT : STRING := '#A-#D-#H #N:#R:#T';
    COLUMN : STRING(40);
    DELTA : UDINT;
  END_VAR
  VAR
    UCB : UNI_CIRCULAR_BUFFER;
    id : WORD;
    delta_last : DT;
  END_VAR

            CASE x.ADD_COM OF

01:	(* ADD INFO *)
	X.ID_MAX := X.ID_MAX + USINT#1;
	id := WORD#16#0D01; (* Quelltype DT , Zieltype STRING *)
02:	(* ADD HEADER *)
	X.UCB.D_STRING := COLUMN;
	X.UCB.D_HEAD := id;
	X.UCB.D_MODE := 1;
	UCB(DATA:=X.UCB); (* Daten eintragen *)
03:	(* ADD DATA *)
	X.UCB.D_STRING := OSCAT_BASIC.DT_TO_STRF(DTI:=X.DTI,MS:=0,FMT:=FMT,LANG:=0);
	X.UCB.D_HEAD := id;
	X.UCB.D_MODE := 1;
	UCB(DATA:=X.UCB); (* Daten eintragen *)
	delta_last := X.DTI;
04:	(* ADD DATA REQ *)
	IF DELTA <> UDINT#0 THEN
		IF DT_TO_UDINT(X.DTI) >= (DT_TO_UDINT(delta_last) + DELTA) THEN
			X.ADD_DATA_REQ := TRUE;
			delta_last := X.DTI;
		END_IF;
	END_IF;
END_CASE;

(* revision history
ks	01. jan. 2011	rev 1.0
	original version

ks	17. may. 2011	rev 1.1
	COLUMN STRING(40), delta

ks	25. july.   2011	rev 1.2
	neue head information

ks	19. apr.   2012	rev 1.3
	code neu überarbeitet
*)
          
END_FUNCTION_BLOCK

FUNCTION_BLOCK DLOG_FILE_TO_FTP
  VAR_IN_OUT
    X : DLOG_DATA;
  END_VAR
  VAR_INPUT
    FTP_URL : STRING(OSCAT_BASIC.STRING_LENGTH);
    FTP_ACTIV : BOOL;
    FILE_DELETE : BOOL;
    TIMEOUT : TIME := TIME#30s0ms;
    RETRY : INT;
    RETRY_TIME : TIME := TIME#30s0ms;
    DNS_IP4 : DWORD;
    PLC_IP4 : DWORD;
  END_VAR
  VAR_OUTPUT
    DONE : BOOL;
    BUSY : BOOL;
    ERROR_C : DWORD;
    ERROR_T : BYTE;
  END_VAR
  VAR
    UCBD : UNI_CIRCULAR_BUFFER_DATA;
    UCB : UNI_CIRCULAR_BUFFER;
    FTP_CLIENT : FTP_CLIENT;
    WT_1 : TON;
    ftrig_old : BOOL;
    filename : STRING;
    step : INT;
    ftp_busy : BOOL;
    ftp_done : BOOL;
    cnt : INT;
  END_VAR

            (* neue Filenamen speichern *)
IF X.NEW_FILE_RTRIG AND ftrig_old = FALSE THEN
	UCBD.D_HEAD := 1;
	UCBD.D_MODE := 1;
	UCBD.D_STRING := X.NEW_FILE;
	UCB(DATA:=UCBD); (* Daten eintragen *)
END_IF;
ftrig_old := X.NEW_FILE_RTRIG;

CASE step OF

00:	IF UCBD.BUF_COUNT > 0 AND ftp_busy = FALSE THEN
		UCBD.D_MODE := 12; (* Daten lesen und löschen *)
		UCB(DATA:=UCBD);
		filename := UCBD.D_STRING;
		cnt := RETRY;
		step := 10;

		(*####################  DEBUG-MESSAGE  ###################################*)
		(*IF _debug_enable THEN
			LOG_CL.NEW_MSG := 'F_T_FTP: Auftrag aktiv /file: ~2';
			LOG_CL.PRINTF[2] := files;
			LOG_MSG();
		END_IF;*)
		(*########################################################################*)

	END_IF;

10:	IF ftp_busy = FALSE THEN
		IF ftp_done THEN
			(*####################  DEBUG-MESSAGE  ###################################*)
			(*IF _debug_enable THEN
				LOG_CL.NEW_MSG := 'F_T_FTP: Auftrag OK /file: ~2';
				LOG_CL.PRINTF[2] := filename;
				LOG_MSG();
			END_IF;*)
			(*########################################################################*)
			step := 0;
		ELSE
			step := 20; (* pause nach error *)
		END_IF;
	END_IF;

20:	IF WT_1.Q THEN (* Wartezeit *)
		cnt := cnt - 1;
		IF RETRY = 0 THEN (* FTP Transfer unbegrenzt wiederholen *)
			(*####################  DEBUG-MESSAGE  ###################################*)
			(*IF _debug_enable THEN
				LOG_CL.NEW_MSG := 'F_T_FTP: Auftrag unbegrenzt wiederholen /file: ~2';
				LOG_CL.PRINTF[2] := filename;
				LOG_MSG();
			END_IF;*)
			(*########################################################################*)
			step := 10; (* FTP Transfer wiederholen *)
		ELSIF cnt >= 0 THEN
			(*####################  DEBUG-MESSAGE  ###################################*)
			(*IF _debug_enable THEN
				LOG_CL.NEW_MSG := 'F_T_FTP: Auftrag wiederholen /cnt: ~1 /file: ~2';
				LOG_CL.PRINTF[1] := INT_TO_STRING(cnt);
				LOG_CL.PRINTF[2] := filename;
				LOG_MSG();
			END_IF;*)
			(*########################################################################*)
			step := 10; (* FTP Transfer wiederholen *)
		ELSE
			(*####################  DEBUG-MESSAGE  ###################################*)
			(*IF _debug_enable THEN
				LOG_CL.NEW_MSG := 'F_T_FTP: Auftrag verworfen /file: ~2';
				LOG_CL.PRINTF[2] := filename;
				LOG_MSG();
			END_IF;*)
			(*########################################################################*)
			step := 0; (* FTP Auftrag verwerfen *)
		END_IF;
	END_IF;

END_CASE;

BUSY := step = 10;
DONE := step = 0;
WT_1(IN:= step = 20, PT:= RETRY_TIME);

FTP_CLIENT(
	ACTIVATE:= BUSY,
	FILENAME:= filename,
	FTP_URL:= FTP_URL,
	FTP_DOWNLOAD:= FALSE,
	FTP_ACTIV:= FTP_ACTIV,
	FILE_DELETE:= FILE_DELETE,
	TIMEOUT:= TIMEOUT,
	DNS_IP4:= DNS_IP4,
	PLC_IP4:= PLC_IP4,
	DONE=> ftp_done,
	BUSY=> ftp_busy
	);

(* Fehlerauswertung *)
IF FTP_CLIENT.ERROR_T <> BYTE#0 THEN
	ERROR_C := FTP_CLIENT.ERROR_C;
	ERROR_T := FTP_CLIENT.ERROR_T;
ELSIF UCBD.BUF_DATA_LOST > UDINT#0 THEN
	ERROR_C := DWORD#2; (* Fehler: Bufferüberlauf - Datenmenge reduzieren *)
	ERROR_T := BYTE#6; 	(* Type: Buffer *)
ELSIF UCBD.BUF_USED_MAX > USINT#90 THEN
	ERROR_C := DWORD#1; (* Warnung: Buffer auslastung > 90% *)
	ERROR_T := BYTE#6;	(* Type: Buffer *)
ELSE
	ERROR_C := DWORD#0;
	ERROR_T := BYTE#0;
END_IF;

(* revision history
ks	01. jan. 2011	rev 1.0
	original version

ks	26. jul. 2011	rev 1.1
    codeoptimierung D_MODE 12

ks	21. mar. 2016	rev 1.2
	fehlermeldungen hinzugefügt
	fehler in RETRY korrigiert
	
*)
          
END_FUNCTION_BLOCK

FUNCTION_BLOCK DLOG_FILE_TO_SMTP
  VAR_IN_OUT
    SERVER : STRING;
    MAILFROM : STRING;
    MAILTO : STRING(OSCAT_BASIC.STRING_LENGTH);
    SUBJECT : STRING;
    BODY : STRING(OSCAT_BASIC.STRING_LENGTH);
    X : DLOG_DATA;
  END_VAR
  VAR_INPUT
    FILE_DELETE : BOOL;
    TIMEOUT : TIME := TIME#30s0ms;
    DTI : DT;
    DTI_OFFSET : INT;
    RETRY : INT;
    RETRY_TIME : TIME := TIME#30s0ms;
    DNS_IP4 : DWORD;
  END_VAR
  VAR_OUTPUT
    DONE : BOOL;
    BUSY : BOOL;
    ERROR_C : DWORD;
    ERROR_T : BYTE;
  END_VAR
  VAR
    UCBD : UNI_CIRCULAR_BUFFER_DATA;
    UCB : UNI_CIRCULAR_BUFFER;
    SMTP_CLIENT : SMTP_CLIENT;
    WT_1 : TON;
    ftrig_old : BOOL;
    files : STRING(OSCAT_BASIC.STRING_LENGTH);
    step : INT;
    smtp_busy : BOOL;
    smtp_done : BOOL;
    cnt : INT;
  END_VAR

            (* neue Filenamen speichern *)
IF X.NEW_FILE_RTRIG AND ftrig_old = FALSE THEN
	UCBD.D_HEAD := 1;
	UCBD.D_MODE := 1;
	UCBD.D_STRING := X.NEW_FILE;
	UCB(DATA:=UCBD); (* Daten eintragen *)
END_IF;
ftrig_old := X.NEW_FILE_RTRIG;

CASE step OF

00:	IF UCBD.BUF_COUNT > 0 AND smtp_busy = FALSE THEN
		UCBD.D_MODE := 12; (* Daten lesen und löschen *)
		UCB(DATA:=UCBD);
		files := UCBD.D_STRING;
		IF FILE_DELETE THEN
			files := CONCAT(files,';#DEL#');
		END_IF;
		cnt := RETRY;
		step := 10;

		(*####################  DEBUG-MESSAGE  ###################################*)
		(*IF _debug_enable THEN
			LOG_CL.NEW_MSG := 'F_T_SMTP: Auftrag aktiv /file: ~2';
			LOG_CL.PRINTF[2] := files;
			LOG_MSG();
		END_IF;*)
		(*########################################################################*)

	END_IF;

10:	IF smtp_busy = FALSE THEN
		IF smtp_done THEN
			(*####################  DEBUG-MESSAGE  ###################################*)
			(*IF _debug_enable THEN
				LOG_CL.NEW_MSG := 'F_T_SMTP: Auftrag OK /file: ~2';
				LOG_CL.PRINTF[2] := files;
				LOG_MSG();
			END_IF;*)
			(*########################################################################*)
			step := 0;
		ELSE
			step := 20; (* pause nach error *)
		END_IF;
	END_IF;

20:	IF WT_1.Q THEN (* Wartezeit *)
		cnt := cnt - 1;
		IF RETRY = 0 THEN (* Transfer unbegrenzt wiederholen *)
			(*####################  DEBUG-MESSAGE  ###################################*)
			(*IF _debug_enable THEN
				LOG_CL.NEW_MSG := 'F_T_SMTP: Auftrag unbegrenzt wiederholen /file: ~2';
				LOG_CL.PRINTF[2] := files;
				LOG_MSG();
			END_IF;*)
			(*########################################################################*)
			step := 10; (* Transfer wiederholen *)
		ELSIF cnt >= 0 THEN
			(*####################  DEBUG-MESSAGE  ###################################*)
			(*IF _debug_enable THEN
				LOG_CL.NEW_MSG := 'F_T_SMTP: Auftrag wiederholen /cnt: ~1 /file: ~2';
				LOG_CL.PRINTF[1] := INT_TO_STRING(cnt);
				LOG_CL.PRINTF[2] := files;
				LOG_MSG();
			END_IF;*)
			(*########################################################################*)
			step := 10; (* Transfer wiederholen *)
		ELSE
			(*####################  DEBUG-MESSAGE  ###################################*)
			(*IF _debug_enable THEN
				LOG_CL.NEW_MSG := 'F_T_SMTP: Auftrag verworfen /file: ~2';
				LOG_CL.PRINTF[2] := files;
				LOG_MSG();
			END_IF;*)
			(*########################################################################*)
			step := 0; (* Auftrag verwerfen *)
		END_IF;
	END_IF;

END_CASE;

BUSY := step = 10;
DONE := step = 0;
WT_1(IN:= step = 20, PT:= RETRY_TIME);

SMTP_CLIENT(
	ACTIVATE:= BUSY,
	TIMEOUT:= TIMEOUT,
	DTI:= DTI,
	DTI_OFFSET:= DTI_OFFSET,
	DNS_IP4:= DNS_IP4,
	SERVER:= SERVER,
	MAILFROM:= MAILFROM,
	MAILTO:= MAILTO,
	SUBJECT:= SUBJECT,
	BODY:= BODY,
	FILES:= FILES,
	DONE=> smtp_done,
	BUSY=> smtp_busy
	);

(* Fehlerauswertung *)
IF SMTP_CLIENT.ERROR_T <> BYTE#0 THEN
	ERROR_C := SMTP_CLIENT.ERROR_C;
	ERROR_T := SMTP_CLIENT.ERROR_T;
ELSIF UCBD.BUF_DATA_LOST > UDINT#0 THEN
	ERROR_C := DWORD#2; (* Fehler: Bufferüberlauf - Datenmenge reduzieren *)
	ERROR_T := BYTE#6; 	(* Type: Buffer *)
ELSIF UCBD.BUF_USED_MAX > USINT#90 THEN
	ERROR_C := DWORD#1; (* Warnung: Buffer auslastung > 90% *)
	ERROR_T := BYTE#6;	(* Type: Buffer *)
ELSE
	ERROR_C := DWORD#0;
	ERROR_T := BYTE#0;
END_IF;

(* revision history

ks	01. jan. 2011	rev 1.0
	original version

ks	28. apr. 2011	rev 1.1
	stringfehler bei option 'file_delete'

ks	26. jul. 2011	rev 1.2
    codeoptimierung D_MODE 12

ks	21. mar. 2016	rev 1.3
	fehlermeldungen hinzugefügt
	fehler in RETRY korrigiert

*)
          
END_FUNCTION_BLOCK

FUNCTION_BLOCK DLOG_REAL
  VAR_IN_OUT
    X : DLOG_DATA;
  END_VAR
  VAR_INPUT
    VALUE : REAL;
    N : INT;
    D : STRING(1) := ',';
    COLUMN : STRING(40);
    DELTA : REAL;
  END_VAR
  VAR
    UCB : UNI_CIRCULAR_BUFFER;
    id : WORD;
    delta_last : REAL;
    value_last : REAL;
  END_VAR

            CASE x.ADD_COM OF

01:	(* ADD INFO *)
	X.ID_MAX := X.ID_MAX + USINT#1;
	id := WORD#16#0201; (* Quelltype REAL , Zieltype STRING *)
02:	(* ADD HEADER *)
	X.UCB.D_STRING := COLUMN;
	X.UCB.D_HEAD := id;
	X.UCB.D_MODE := 1;
	UCB(DATA:=X.UCB); (* Daten eintragen *)
03:	(* ADD DATA *)
	X.UCB.D_STRING := OSCAT_BASIC.REAL_TO_STRF(IN:=value_last,N:=N,D:=D);
	X.UCB.D_HEAD := id;
	X.UCB.D_MODE := 1;
	UCB(DATA:=X.UCB); (* Daten eintragen *)
	delta_last := value_last;
04:	(* ADD DATA REQ *)
	IF DELTA <> 0.0 THEN
		IF VALUE <= (delta_last - DELTA) OR VALUE >= (delta_last + DELTA) THEN
			X.ADD_DATA_REQ := TRUE;
			delta_last := VALUE;
		END_IF;
	END_IF;
END_CASE;
value_last := VALUE;

(* revision history
ks	01. jan. 2011	rev 1.0
	original version

ks	17. may. 2011	rev 1.1
	DELTA Funktion integriert

ks	25. july.   2011	rev 1.2
	neue head information

ks	19. apr.   2012	rev 1.3
	code neu überarbeitet
*)
          
END_FUNCTION_BLOCK

FUNCTION_BLOCK DLOG_REAL_ARRAY
  VAR_IN_OUT
    R_ARRAY : DLOG_REAL_ARRAY_DATA;
    X : DLOG_DATA;
  END_VAR
  VAR_INPUT
    N : INT;
    D : STRING(1);
    R_COUNT : INT;
  END_VAR
  VAR
    UCB : UNI_CIRCULAR_BUFFER;
    id : WORD;
    idx : INT;
  END_VAR

            FOR idx := 1 TO R_COUNT DO

	CASE x.ADD_COM OF

	01:	(* ADD INFO *)
		X.ID_MAX := X.ID_MAX + USINT#1;
		id := WORD#16#0201; (* Quelltype REAL , Zieltype STRING *)
		(* automatisch Namen vergeben *)
		IF LEN(R_ARRAY[idx].COLUMN) = 0 THEN
			R_ARRAY[idx].COLUMN := CONCAT('Spalte_',USINT_TO_STRING(X.ID_MAX));
		END_IF;
	02:	(* ADD HEADER *)
		X.UCB.D_STRING := R_ARRAY[idx].COLUMN;
		X.UCB.D_HEAD := id;
		X.UCB.D_MODE := 1;
		UCB(DATA:=X.UCB); (* Daten eintragen *)
	03:	(* ADD DATA *)
		X.UCB.D_STRING := OSCAT_BASIC.REAL_TO_STRF(IN:=R_ARRAY[idx]._value_last,N:=N,D:=D);
		X.UCB.D_HEAD := id;
		X.UCB.D_MODE := 1;
		UCB(DATA:=X.UCB); (* Daten eintragen *)
		R_ARRAY[idx]._delta_last := R_ARRAY[idx]._value_last;
	04:	(* ADD DATA REQ *)
		IF R_ARRAY[idx].DELTA <> 0.0 THEN
			IF R_ARRAY[idx].VALUE <= (R_ARRAY[idx]._delta_last - R_ARRAY[idx].DELTA) OR R_ARRAY[idx].VALUE >= (R_ARRAY[idx]._delta_last + R_ARRAY[idx].DELTA) THEN
				X.ADD_DATA_REQ := TRUE;
				R_ARRAY[idx]._delta_last := R_ARRAY[idx].VALUE;
			END_IF;
		END_IF;
	END_CASE;
	R_ARRAY[idx]._value_last := R_ARRAY[idx].VALUE;

END_FOR;

(* revision history
ks	03. mar. 2016	rev 1.0
	original version

*)
          
END_FUNCTION_BLOCK

FUNCTION_BLOCK DLOG_STORE_FILE_CSV
  VAR_IN_OUT
    X : DLOG_DATA;
    SAVE_DATA : DLOG_SAVE;
  END_VAR
  VAR_INPUT
    ENABLE : BOOL;
    TRIG_M : BOOL;
    TRIG_T : TIME;
    FILENAME : STRING;
    DTI : DT;
    SEP : BYTE;
    AUTO_CLOSE : TIME := TIME#15s0ms;
  END_VAR
  VAR_OUTPUT
    ERROR_C : DWORD;
    ERROR_T : BYTE;
  END_VAR
  VAR
    FS : FILE_SERVER;
    FSD : FILE_SERVER_DATA;
    PT : NETWORK_BUFFER;
    UCB : UNI_CIRCULAR_BUFFER;
    trig_auto : BOOL;
    trig_stored : BOOL;
    trig_tmp : BOOL;
    trig_m_last : BOOL;
    dti_last : DT := DATE_AND_TIME#2070-2-6-6:28:15;
    fn_last : STRING;
    fn : STRING;
    step_1 : INT;
    step_2 : INT;
    idx : INT;
    log_stop : BOOL;
    n : USINT;
    wd_ton : TON;
    wd_time : TIME;
    aw_ton : TON;
    aw_enable : BOOL;
    aw_aktiv : BOOL;
    total_bytes : UDINT;
  END_VAR

            X.DTI := DTI; (* Datum / Zeit eintragen *)
X.CLOCK_TRIG := DTI <> dti_last;
dti_last := DTI;
trig_auto := FALSE;
IF X.CLOCK_TRIG THEN (* Impuls in jeder Sekunde *)
	fn := OSCAT_BASIC.DT_TO_STRF(DTI, 0, FILENAME, 0); (* automatische Dateinamen generierung *)
	IF TRIG_T >= T#1000ms THEN (* automatischer Trigger *)
		trig_auto := DT_TO_UDINT(DTI) MOD (TIME_TO_UDINT(TRIG_T) / UDINT#1000) = UDINT#0;
	END_IF;
END_IF;

CASE step_1 OF

00:	IF ENABLE THEN
		aw_enable := AUTO_CLOSE >= T#5s;
		wd_time := SEL(X.LOAD_TIME_MAX > T#0s, T#5ms,X.LOAD_TIME_MAX);
		fn_last := fn; (* aktuellen Dateinnamen speichern *)
		IF X.ID_MAX = USINT#0 THEN (* nur einmal nach Satellitenbausteinen scannen *)
			X.ADD_COM := 01; (* ADD INFO *)
			X.STORE_TYPE := BYTE#2; (* CSV-Modus *)
		END_IF;
		step_1 := 10;

		(* ---------------- Debug-Message -----------------------*)
		(*IF _debug_enable THEN
			LOG_CL.NEW_MSG := 'FILE_CSV1 - Start: File [~1], [~2]';
			LOG_CL.PRINTF[1] := fn_last;
			LOG_CL.PRINTF[2] := DT_TO_STRING(DTI);
			LOG_MSG();
		END_IF;*)
		(* -----------------------------------------------------------------*)

	END_IF;

10:	X.UCB.D_STRING := fn_last;
	IF fn_last = SAVE_DATA.FN_REM THEN
		X.UCB.D_HEAD := WORD#16#F201; (* Filemode open + write *)
		X.ADD_COM := 00;
	ELSE
		X.UCB.D_HEAD := WORD#16#F301; (* Filemode create + write *)
		X.ADD_COM := 02; (* ADD HEADER *)
	END_IF;

	X.UCB.D_MODE := 1; (* Dateinamen als String ablegen *)
	UCB(DATA:=X.UCB); (* Daten eintragen *)
	step_1 := 30;

30:	(* LOG-Trigger verarbeiten *)
	trig_tmp := (TRIG_M AND NOT trig_m_last) OR trig_auto OR X.ADD_DATA_REQ;

	IF ENABLE = FALSE OR fn <> fn_last THEN (* ENABLE = 0 oder neuen Dateinamen -> Log Stop *)
		trig_stored := trig_tmp; (* aktuellen Triggerpuls speichern *)
		X.UCB.D_HEAD := WORD#16#EE00;
		X.UCB.D_MODE := 1;
		UCB(DATA:=X.UCB); (* Element schreiben *)
		X.ADD_COM := 00;
		step_1 := 00;

		(* ---------------- Debug-Message -----------------------*)
		(*IF _debug_enable THEN
			LOG_CL.NEW_MSG := 'FILE_CSV1 - Stop: [~2]';
			LOG_CL.PRINTF[2] := DT_TO_STRING(DTI);
			LOG_MSG();
		END_IF;*)
		(* -----------------------------------------------------------------*)

	ELSIF ENABLE THEN
		IF trig_tmp OR trig_stored THEN (* manueller, automatischer oder externer Trigger *)
			trig_stored := FALSE;
			X.ADD_COM := 03; (* ADD DATA *)
			SAVE_DATA.TRIG_CNT := SAVE_DATA.TRIG_CNT + UDINT#1;
			SAVE_DATA.TRIG_CNT_TOTAL  := SAVE_DATA.TRIG_CNT_TOTAL + UDINT#1;
			(* ---------------- Debug-Message -----------------------*)
			(*IF _debug_enable THEN
				LOG_CL.NEW_MSG := 'FILE_CSV1 - Trig: [~2]';
				LOG_CL.PRINTF[2] := DT_TO_STRING(DTI);
				LOG_MSG();
			END_IF;*)
			(* -----------------------------------------------------------------*)
		ELSE
			X.ADD_COM := 04;	(* ADD DATA REQ *)
		END_IF;
	END_IF;

END_CASE;
X.ADD_DATA_REQ := FALSE; (* externe Anforderung rücksetzen *)

(* ##################################### *)

CASE step_2 OF

00:	aw_ton(IN:= idx > 0 AND aw_enable, PT:= AUTO_CLOSE); (* AutoWrite Timer *)
	IF aw_ton.Q THEN (* Zeitgesteuertes Datenschreiben *)
		aw_aktiv := TRUE;
		step_2 := 10; (* Daten schreiben *)
		(* ---------------- Debug-Message -----------------------*)
		(*IF _debug_enable THEN
			LOG_CL.NEW_MSG := 'FILE_CSV2 - AutoWrite: [~2]';
			LOG_CL.PRINTF[2] := DT_TO_STRING(DTI);
			LOG_MSG();
		END_IF;*)
		(* -----------------------------------------------------------------*)

	ELSE
		wd_ton(IN:= FALSE, PT:= wd_time);
		wd_ton(IN:= TRUE);
		WHILE X.UCB.BUF_COUNT > 0 AND step_2 = 0 AND wd_ton.Q = FALSE DO

			X.UCB.D_MODE := 10;
			UCB(DATA:=X.UCB); (* Element lesen , aber noch nicht entfernen *)
			IF X.UCB.D_HEAD > WORD#16#F000 THEN (* F301 oder F201 *)
				X.UCB.D_MODE := 11;
				UCB(DATA:=X.UCB); (* Element entfernen *)
	
				FSD.MODE := WORD_TO_BYTE(SHR(SHL(X.UCB.D_HEAD,4),12)); (* 0X00 -> 000X = 3 create + write / 2 open + write *)
				FSD.OFFSET := UDINT#0; (* Start bei Dateianfang *)
				FSD.FILENAME := X.UCB.D_STRING; (* Dateiname *)
				PT.SIZE := UINT#0;
				SAVE_DATA.FN_REM := FSD.FILENAME; (* aktuellen Dateinamen remanent sichern *)
	
				IF FSD.MODE = BYTE#3 THEN	(* Datei neu anlegen -> dann zähler reset *)
					SAVE_DATA.TRIG_CNT := UDINT#0;
				END_IF;
	
				X.NEW_FILE := FSD.FILENAME;
				X.NEW_FILE_SIZE := UDINT#0;
				X.NEW_FILE_RTRIG := FALSE;
				step_2 := 20;
				(* ---------------- Debug-Message -----------------------*)
				(*IF _debug_enable THEN
					LOG_CL.NEW_MSG := 'FILE_CSV2 - Create: Mode [~1] , [~2]';
					LOG_CL.PRINTF[2] := DT_TO_STRING(DTI);
					LOG_CL.PRINTF[1] := BYTE_TO_STRING(FSD.MODE);
					LOG_MSG();
				END_IF;*)
				(* -----------------------------------------------------------------*)

			ELSIF X.UCB.D_HEAD = WORD#16#EE00 THEN (* LOG_STOP Command *)
				X.UCB.D_MODE := 11;
				UCB(DATA:=X.UCB); (* Element entfernen *)
				log_stop := TRUE;
				step_2 := 10; (* Daten schreiben *)

			ELSIF idx + X.UCB.D_SIZE + 2 < SIZEOF(PT.BUFFER) THEN (* bufferplatz vorhanden *)
				X.UCB.D_MODE := 11;
				UCB(DATA:=X.UCB); (* Element entfernen *)
				(* ---------------- Debug-Message -----------------------*)
				(*IF _debug_enable THEN
					LOG_CL.NEW_MSG := 'FILE_CSV2 - BUF: TXT [~1],Pos [~2], [~3]';
					LOG_CL.PRINTF[1] := X.UCB.D_STRING;
					LOG_CL.PRINTF[2] := INT_TO_STRING(idx);
					LOG_CL.PRINTF[3] := DT_TO_STRING(DTI);
					LOG_MSG();
				END_IF;*)
				(* -----------------------------------------------------------------*)
				OSCAT_BASIC._STRING_TO_BUFFER(STR:=X.UCB.D_STRING, POS:=idx, PT:=ADR(PT.BUFFER), SIZE:=SIZEOF(PT.BUFFER));
				idx := idx + LEN(X.UCB.D_STRING);
				n := n + USINT#1;
				IF n = X.ID_MAX THEN (* letztes Element einer Zeile *)
					n := USINT#0;
					PT.BUFFER[idx] := BYTE#16#0D;
					idx := idx + 1;
					PT.BUFFER[idx] := BYTE#16#0A;
				ELSE
					PT.BUFFER[idx] := SEP;
				END_IF;
				idx := idx + 1;
				X.NEW_FILE_SIZE := total_bytes + INT_TO_UDINT(idx);
			ELSE (* kein Platz vorhanden *)
				step_2 := 10; (* Daten schreiben *)
			END_IF;
			wd_ton();
		END_WHILE;
	END_IF;

10:	IF idx > 0 THEN (* Daten schreiben *)
		FSD.MODE := BYTE#2; (* File_Open_Exist + File_Write *)
		FSD.OFFSET := UDINT#4294967294; (* 16#FFFF_FFFE ->Spezialcode: Daten automatisch an Dateiende anhängen *)
		PT.SIZE := INT_TO_UINT(idx); (* Datenlänge eintragen *)
		idx := 0;
		(* ---------------- Debug-Message -----------------------*)
		(*IF _debug_enable THEN
			LOG_CL.NEW_MSG := 'FILE_CSV2 - WriteData: Mode [~3] Size [~1] , [~2]';
			LOG_CL.PRINTF[1] := UINT_TO_STRING(PT.SIZE);
			LOG_CL.PRINTF[2] := DT_TO_STRING(DTI);
			LOG_CL.PRINTF[3] := BYTE_TO_STRING(FSD.MODE);
			LOG_MSG();
		END_IF;*)
		(* -----------------------------------------------------------------*)
	END_IF;
	step_2 := 20;

20:	IF FSD.MODE = BYTE#0 THEN
		total_bytes := FSD.FILE_SIZE;
		X.NEW_FILE_SIZE := total_bytes + INT_TO_UDINT(idx);
		IF log_stop OR aw_aktiv THEN
			aw_aktiv := FALSE;
			FSD.MODE := BYTE#5; (* Datei schliessen *)
			(* ---------------- Debug-Message -----------------------*)
			(*IF _debug_enable THEN
				LOG_CL.NEW_MSG := 'FILE_CSV2 - Close: [~2]';
				LOG_CL.PRINTF[2] := DT_TO_STRING(DTI);
				LOG_MSG();
			END_IF;*)
			(* -----------------------------------------------------------------*)
		END_IF;
		step_2 := 30;
	END_IF;

30:	IF FSD.MODE = BYTE#0 THEN (* Befehl beendet ? *)
		IF log_stop THEN
			X.NEW_FILE_RTRIG := TRUE;
			log_stop := FALSE;
			SAVE_DATA.FN_REM := ''; (* remanenten Dateinamen löschen *)
		END_IF;
		step_2 := 00;
	END_IF;

END_CASE;

FS(FSD:=FSD,PT:=PT); (* FILE_SERVER *)
(* Fehlerauswertung *)
IF FSD.ERROR <> BYTE#0 THEN
	ERROR_C := BYTE_TO_DWORD(FSD.ERROR);
	ERROR_T := BYTE#1;
ELSIF X.UCB.BUF_DATA_LOST > UDINT#0 THEN
	ERROR_C := DWORD#2; (* Fehler: Bufferüberlauf - Datenmenge reduzieren *)
	ERROR_T := BYTE#6; 	(* Type: Buffer *)
ELSIF X.UCB.BUF_USED_MAX > USINT#90 THEN
	ERROR_C := DWORD#1; (* Warnung: Buffer auslastung > 90% *)
	ERROR_T := BYTE#6;	(* Type: Buffer *)
ELSE
	ERROR_C := DWORD#0;
	ERROR_T := BYTE#0;
END_IF;

trig_m_last := TRIG_M;

(* revision history
ks	01. jan. 2011	rev 1.0
	original version

ks	13. may. 2011	rev 1.1
	ADD_DATA_REQ, ERROR_T, ERROR_C hinzugefügt

ks	25. july. 2011	rev 1.2
	HEAD Informationen geändert, neuer Spaltenzähler

ks	16. apr. 2012	rev 1.3
	neuer überarbeiteter Code für automatisches File-open/close

ks	8. mar. 2016	rev 1.4
	nur einmal nach satellitenbausteinen scannen

ks	21. mar. 2016	rev 1.5
	prüfung auf freien bufferplatz hinzugefügt
	fehlermeldungen hinzugefügt
*)
          
END_FUNCTION_BLOCK

FUNCTION_BLOCK DLOG_STORE_FILE_HTML
  VAR_IN_OUT
    X : DLOG_DATA;
    SAVE_DATA : DLOG_SAVE;
  END_VAR
  VAR_INPUT
    ENABLE : BOOL;
    TRIG_M : BOOL;
    TRIG_T : TIME;
    FILENAME : STRING;
    DTI : DT;
    AUTO_CLOSE : TIME := TIME#15s0ms;
    HTML_CAPTION : STRING;
    HTML_TABLE : STRING;
    HTML_TR_HEAD : STRING;
    HTML_TR_EVEN : STRING;
    HTML_TR_ODD : STRING;
  END_VAR
  VAR_OUTPUT
    ERROR_C : DWORD;
    ERROR_T : BYTE;
  END_VAR
  VAR
    FS : FILE_SERVER;
    FSD : FILE_SERVER_DATA;
    PT : NETWORK_BUFFER;
    UCB : UNI_CIRCULAR_BUFFER;
    trig_auto : BOOL;
    trig_stored : BOOL;
    trig_tmp : BOOL;
    trig_m_last : BOOL;
    dti_last : DT := DATE_AND_TIME#2070-2-6-6:28:15;
    fn_last : STRING;
    str : STRING(OSCAT_BASIC.STRING_LENGTH);
    fn : STRING;
    step_1 : INT;
    step_2 : INT;
    idx : INT;
    log_state : USINT;
    log_stop : BOOL;
    n : INT;
    wd_ton : TON;
    wd_time : TIME;
    aw_ton : TON;
    aw_enable : BOOL;
    aw_aktiv : BOOL;
    total_bytes : UDINT;
    cur_ode : BYTE;
  END_VAR

            X.DTI := DTI; (* Datum / Zeit eintragen *)
X.CLOCK_TRIG := DTI <> dti_last;
dti_last := DTI;
trig_auto := FALSE;
IF X.CLOCK_TRIG THEN (* Impuls in jeder Sekunde *)
	fn := OSCAT_BASIC.DT_TO_STRF(DTI, 0, FILENAME, 0); (* automatische Dateinamen generierung *)
	IF TRIG_T >= T#1000ms THEN (* automatischer Trigger *)
		trig_auto := DT_TO_UDINT(DTI) MOD (TIME_TO_UDINT(TRIG_T) / UDINT#1000) = UDINT#0;
	END_IF;
END_IF;

CASE step_1 OF

00:	IF ENABLE THEN
		aw_enable := AUTO_CLOSE >= T#5s;
		wd_time := SEL(X.LOAD_TIME_MAX > T#0s, T#5ms,X.LOAD_TIME_MAX);
		fn_last := fn; (* aktuellen Dateinnamen speichern *)
		IF X.ID_MAX = USINT#0 THEN (* nur einmal nach Satellitenbausteinen scannen *)
			X.ADD_COM := 01; (* ADD INFO *)
			X.STORE_TYPE := BYTE#4; (* HTML-Modus *)
		END_IF;
		step_1 := 10;

		(* ---------------- Debug-Message -----------------------*)
		(*IF _debug_enable THEN
			LOG_CL.NEW_MSG := 'FILE_HTML1 - Start: File [~1], [~2]';
			LOG_CL.PRINTF[1] := fn_last;
			LOG_CL.PRINTF[2] := DT_TO_STRING(DTI);
			LOG_MSG();
		END_IF;*)
		(* -----------------------------------------------------------------*)

	END_IF;

10:	X.UCB.D_STRING := fn_last;
	IF fn_last = SAVE_DATA.FN_REM THEN
		X.UCB.D_HEAD := WORD#16#F201; (* Filemode open + write *)
		X.ADD_COM := 00;
	ELSE
		X.UCB.D_HEAD := WORD#16#F301; (* Filemode create + write *)
		X.ADD_COM := 02; (* ADD HEADER *)
	END_IF;

	X.UCB.D_MODE := 1; (* Dateinamen als String ablegen *)
	UCB(DATA:=X.UCB); (* Daten eintragen *)
	step_1 := 30;

30:	(* LOG-Trigger verarbeiten *)
	trig_tmp := (TRIG_M AND NOT trig_m_last) OR trig_auto OR X.ADD_DATA_REQ;

	IF ENABLE = FALSE OR fn <> fn_last THEN (* ENABLE = 0 oder neuen Dateinamen -> Log Stop *)
		trig_stored := trig_tmp; (* aktuellen Triggerpuls speichern *)
		X.UCB.D_HEAD := WORD#16#EE00;
		X.UCB.D_MODE := 1;
		UCB(DATA:=X.UCB); (* Element schreiben *)
		X.ADD_COM := 00;
		step_1 := 00;

		(* ---------------- Debug-Message -----------------------*)
		(*IF _debug_enable THEN
			LOG_CL.NEW_MSG := 'FILE_HTML1 - Stop: [~2]';
			LOG_CL.PRINTF[2] := DT_TO_STRING(DTI);
			LOG_MSG();
		END_IF;*)
		(* -----------------------------------------------------------------*)

	ELSIF ENABLE THEN
		IF trig_tmp OR trig_stored THEN (* manueller, automatischer oder externer Trigger *)
			trig_stored := FALSE;
			X.ADD_COM := 03; (* ADD DATA *)
			SAVE_DATA.TRIG_CNT := SAVE_DATA.TRIG_CNT + UDINT#1;
			SAVE_DATA.TRIG_CNT_TOTAL  := SAVE_DATA.TRIG_CNT_TOTAL + UDINT#1;
			(* ---------------- Debug-Message -----------------------*)
			(*IF _debug_enable THEN
				LOG_CL.NEW_MSG := 'FILE_HTML1 - Trig: [~2]';
				LOG_CL.PRINTF[2] := DT_TO_STRING(DTI);
				LOG_MSG();
			END_IF;*)
			(* -----------------------------------------------------------------*)
		ELSE
			X.ADD_COM := 04;	(* ADD DATA REQ *)
		END_IF;
	END_IF;

END_CASE;
X.ADD_DATA_REQ := FALSE; (* externe Anforderung rücksetzen *)

(* ##################################### *)

CASE step_2 OF

00:	aw_ton(IN:= idx > 0 AND aw_enable , PT:= AUTO_CLOSE); (* AutoWrite Timer *)
	IF aw_ton.Q THEN (* Zeitgesteuertes Datenschreiben *)
		aw_aktiv := TRUE;
		step_2 := 10; (* Daten schreiben *)
		(* ---------------- Debug-Message -----------------------*)
		(*IF _debug_enable THEN
			LOG_CL.NEW_MSG := 'FILE_HTML2 - AutoWrite: [~2]';
			LOG_CL.PRINTF[2] := DT_TO_STRING(DTI);
			LOG_MSG();
		END_IF;*)
		(* -----------------------------------------------------------------*)

	ELSE
		wd_ton(IN:= FALSE, PT:= wd_time);
		wd_ton(IN:= TRUE);
		WHILE X.UCB.BUF_COUNT > 0 AND step_2 = 0 AND wd_ton.Q = FALSE DO

			X.UCB.D_MODE := 10;
			UCB(DATA:=X.UCB); (* Element lesen , aber noch nicht entfernen *)

			IF X.UCB.D_HEAD > WORD#16#F000 THEN (* F301 oder F201 *)

				str := CONCAT('<html><body><table ',HTML_TABLE);
		        		str := CONCAT(str,'><caption>');
		        		str := CONCAT(str,HTML_CAPTION);
		        		str := CONCAT(str,'</caption>');

				IF idx + LEN(str) < SIZEOF(PT.BUFFER) THEN (* Platz für Element vorhanden ? *)

					FSD.MODE := WORD_TO_BYTE(SHR(SHL(X.UCB.D_HEAD,4),12)); (* 0X00 -> 000X = 3 create + write / 2 open + write *)
					FSD.OFFSET := UDINT#0; (* Start bei Dateianfang *)
					FSD.FILENAME := X.UCB.D_STRING; (* Dateiname *)
					PT.SIZE := UINT#0;
					SAVE_DATA.FN_REM := FSD.FILENAME; (* aktuellen Dateinamen remanent sichern *)

					X.NEW_FILE := FSD.FILENAME;
					X.NEW_FILE_SIZE := UDINT#0;
					X.NEW_FILE_RTRIG := FALSE;
					step_2 := 20;
	
					(* Headerdaten schreiben *)
					IF FSD.MODE = BYTE#3 THEN
						SAVE_DATA.TRIG_CNT := UDINT#0; (* Datei neu anlegen -> dann zähler reset *)
						SAVE_DATA.COLOR := FALSE;
						SAVE_DATA.HEAD := FALSE;

						OSCAT_BASIC._STRING_TO_BUFFER(STR:=str, POS:=idx, PT:=ADR(PT.BUFFER), SIZE:=SIZEOF(PT.BUFFER));
						idx := idx + LEN(str);
						X.NEW_FILE_SIZE := total_bytes + INT_TO_UDINT(idx);
					END_IF;

					X.UCB.D_MODE := 11;
					UCB(DATA:=X.UCB); (* Element entfernen *)

					(* ---------------- Debug-Message -----------------------*)
					(*IF _debug_enable THEN
						LOG_CL.NEW_MSG := 'FILE_HTML2 - Create: Mode [~1] , [~2]';
						LOG_CL.PRINTF[2] := DT_TO_STRING(DTI);
						LOG_CL.PRINTF[1] := BYTE_TO_STRING(FSD.MODE);
						LOG_MSG();
					END_IF;*)
					(* -----------------------------------------------------------------*)
				END_IF;

			ELSIF X.UCB.D_HEAD = WORD#16#EE00 THEN (* LOG_STOP Command *)

				str := '</table></body></html>';

				IF idx + LEN(str) < SIZEOF(PT.BUFFER) THEN (* Platz für Element vorhanden ? *)

					OSCAT_BASIC._STRING_TO_BUFFER(STR:=str, POS:=idx, PT:=ADR(PT.BUFFER), SIZE:=SIZEOF(PT.BUFFER));
					idx := idx + LEN(str);
					log_stop := TRUE;
					step_2 := 10; (* Daten schreiben *)

					X.UCB.D_MODE := 11;
					UCB(DATA:=X.UCB); (* Element entfernen *)
				END_IF;

			ELSIF idx + LEN(X.UCB.D_STRING) + 120 < SIZEOF(PT.BUFFER) THEN (* Platz für Element vorhanden ? *)

				(* ---------------- Debug-Message -----------------------*)
				(*IF _debug_enable THEN
					LOG_CL.NEW_MSG := 'FILE_CSV2 - BUF: TXT [~1],Pos [~2], [~3]';
					LOG_CL.PRINTF[1] := X.UCB.D_STRING;
					LOG_CL.PRINTF[2] := INT_TO_STRING(idx);
					LOG_CL.PRINTF[3] := DT_TO_STRING(DTI);
					LOG_MSG();
				END_IF;*)
				(* -----------------------------------------------------------------*)

				IF log_state = USINT#0 THEN
					str := '<TR ';
					IF NOT SAVE_DATA.HEAD THEN
						str := CONCAT(str,HTML_TR_HEAD);
						SAVE_DATA.HEAD := TRUE;
					ELSIF SAVE_DATA.COLOR THEN
						str := CONCAT(str,HTML_TR_EVEN);
					ELSE
						str := CONCAT(str,HTML_TR_ODD);
					END_IF;
					str := CONCAT(str,'><TD>');
				ELSE
					str := '<TD>';
				END_IF;

				OSCAT_BASIC._STRING_TO_BUFFER(STR:=str, POS:=idx, PT:=ADR(PT.BUFFER), SIZE:=SIZEOF(PT.BUFFER));
				idx := idx + LEN(str);
				log_state := log_state + USINT#1;

				OSCAT_BASIC._STRING_TO_BUFFER(STR:=X.UCB.D_STRING, POS:=idx, PT:=ADR(PT.BUFFER), SIZE:=SIZEOF(PT.BUFFER));
				idx := idx + LEN(X.UCB.D_STRING);
				n := n + USINT#1;
				IF n >= X.ID_MAX THEN
					n := USINT#0;
					str := '</TD></TR>';
					SAVE_DATA.COLOR := NOT SAVE_DATA.COLOR;
					log_state := USINT#0;
				ELSE
					str := '</TD>';
				END_IF;
				OSCAT_BASIC._STRING_TO_BUFFER(STR:=str, POS:=idx, PT:=ADR(PT.BUFFER), SIZE:=SIZEOF(PT.BUFFER));
				idx := idx + LEN(str);
				X.NEW_FILE_SIZE := total_bytes + INT_TO_UDINT(idx);

				X.UCB.D_MODE := 11;
				UCB(DATA:=X.UCB); (* Element entfernen *)

			ELSE (* kein Platz vorhanden *)
				step_2 := 10; (* Daten schreiben *)

			END_IF;
			wd_ton();
		END_WHILE;
	END_IF;

10:	IF idx > 0 THEN (* Daten schreiben *)
		FSD.MODE := BYTE#2; (* File_Open_Exist + File_Write *)
		FSD.OFFSET := UDINT#4294967294; (* 16#FFFF_FFFE ->Spezialcode: Daten automatisch an Dateiende anhängen *)
		PT.SIZE := INT_TO_UINT(idx); (* Datenlänge eintragen *)
		idx := 0;
		(* ---------------- Debug-Message -----------------------*)
		(*IF _debug_enable THEN
			LOG_CL.NEW_MSG := 'FILE_HTML2 - WriteData: Mode [~3] Size [~1] , [~2]';
			LOG_CL.PRINTF[1] := UINT_TO_STRING(PT.SIZE);
			LOG_CL.PRINTF[2] := DT_TO_STRING(DTI);
			LOG_CL.PRINTF[3] := BYTE_TO_STRING(FSD.MODE);
			LOG_MSG();
		END_IF;*)
		(* -----------------------------------------------------------------*)
	END_IF;
	step_2 := 20;

20:	IF FSD.MODE = BYTE#0 THEN
		total_bytes := FSD.FILE_SIZE;
		X.NEW_FILE_SIZE := total_bytes + INT_TO_UDINT(idx);
		IF log_stop OR aw_aktiv THEN
			aw_aktiv := FALSE;
			FSD.MODE := BYTE#5; (* Datei schliessen *)
			(* ---------------- Debug-Message -----------------------*)
			(*IF _debug_enable THEN
				LOG_CL.NEW_MSG := 'FILE_HTML2 - Close: [~2]';
				LOG_CL.PRINTF[2] := DT_TO_STRING(DTI);
				LOG_MSG();
			END_IF;*)
			(* -----------------------------------------------------------------*)
		END_IF;
		step_2 := 30;
	END_IF;

30:	IF FSD.MODE = BYTE#0 THEN (* Datei schliessen beendet *)
		IF log_stop THEN
			X.NEW_FILE_RTRIG := TRUE;
			log_stop := FALSE;
			SAVE_DATA.FN_REM := ''; (* remanenten Dateinamen löschen *)
		END_IF;
		step_2 := 00;
	END_IF;

END_CASE;

FS(FSD:=FSD,PT:=PT); (* FILE_SERVER *)

(* Fehlerauswertung *)
IF FSD.ERROR <> BYTE#0 THEN
	ERROR_C := BYTE_TO_DWORD(FSD.ERROR);
	ERROR_T := BYTE#1;
ELSIF X.UCB.BUF_DATA_LOST > UDINT#0 THEN
	ERROR_C := DWORD#2; (* Fehler: Bufferüberlauf - Datenmenge reduzieren *)
	ERROR_T := BYTE#6; 	(* Type: Buffer *)
ELSIF X.UCB.BUF_USED_MAX > USINT#90 THEN
	ERROR_C := DWORD#1; (* Warnung: Buffer auslastung > 90% *)
	ERROR_T := BYTE#6;	(* Type: Buffer *)
ELSE
	ERROR_C := DWORD#0;
	ERROR_T := BYTE#0;
END_IF;

trig_m_last := TRIG_M;

(* revision history
ks	25. july. 2011	rev 1.0
	original version

ks	16. apr. 2012	rev 1.1
	neuer überarbeiteter Code für automatisches File-open/close

ks	8. mar. 2016	rev 1.2
	nur einmal nach satellitenbausteinen scannen

ks	21. mar. 2016	rev 1.3
	prüfung auf freien bufferplatz hinzugefügt
	fehlermeldungen hinzugefügt

*)
          
END_FUNCTION_BLOCK

FUNCTION_BLOCK DLOG_STORE_FILE_XML
  VAR_IN_OUT
    X : DLOG_DATA;
    SAVE_DATA : DLOG_SAVE;
  END_VAR
  VAR_INPUT
    ENABLE : BOOL;
    TRIG_M : BOOL;
    TRIG_T : TIME;
    FILENAME : STRING;
    DTI : DT;
    AUTO_CLOSE : TIME := TIME#15s0ms;
  END_VAR
  VAR_OUTPUT
    ERROR_C : DWORD;
    ERROR_T : BYTE;
  END_VAR
  VAR
    FS : FILE_SERVER;
    FSD : FILE_SERVER_DATA;
    PT : NETWORK_BUFFER;
    UCB : UNI_CIRCULAR_BUFFER;
    trig_auto : BOOL;
    trig_stored : BOOL;
    trig_tmp : BOOL;
    trig_m_last : BOOL;
    dti_last : DT := DATE_AND_TIME#2070-2-6-6:28:15;
    fn_last : STRING;
    fn : STRING;
    str : STRING(OSCAT_BASIC.STRING_LENGTH);
    step_1 : INT;
    step_2 : INT;
    idx : INT;
    log_state : USINT;
    log_stop : BOOL;
    n : INT;
    wd_ton : TON;
    wd_time : TIME;
    aw_ton : TON;
    aw_enable : BOOL;
    aw_aktiv : BOOL;
    total_bytes : UDINT;
  END_VAR

            X.DTI := DTI; (* Datum / Zeit eintragen *)
X.CLOCK_TRIG := DTI <> dti_last;
dti_last := DTI;
trig_auto := FALSE;
IF X.CLOCK_TRIG THEN (* Impuls in jeder Sekunde *)
	fn := OSCAT_BASIC.DT_TO_STRF(DTI, 0, FILENAME, 0); (* automatische Dateinamen generierung *)
	IF TRIG_T >= T#1000ms THEN (* automatischer Trigger *)
		trig_auto := DT_TO_UDINT(DTI) MOD (TIME_TO_UDINT(TRIG_T) / UDINT#1000) = UDINT#0;
	END_IF;
END_IF;

CASE step_1 OF

00:	IF ENABLE THEN
		aw_enable := AUTO_CLOSE >= T#5s;
		wd_time := SEL(X.LOAD_TIME_MAX > T#0s, T#5ms,X.LOAD_TIME_MAX);
		fn_last := fn; (* aktuellen Dateinnamen speichern *)
		IF X.ID_MAX = USINT#0 THEN (* nur einmal nach Satellitenbausteinen scannen *)
			X.ADD_COM := 01; (* ADD INFO *)
			X.STORE_TYPE := BYTE#3; (* XML-Modus *)
		END_IF;
		step_1 := 10;

		(* ---------------- Debug-Message -----------------------*)
		(*IF _debug_enable THEN
			LOG_CL.NEW_MSG := 'FILE_XML1 - Start: File [~1], [~2]';
			LOG_CL.PRINTF[1] := fn_last;
			LOG_CL.PRINTF[2] := DT_TO_STRING(DTI);
			LOG_MSG();
		END_IF;*)
		(* -----------------------------------------------------------------*)

	END_IF;

10:	X.UCB.D_STRING := fn_last;
	IF fn_last = SAVE_DATA.FN_REM THEN
		X.UCB.D_HEAD := WORD#16#F201; (* Filemode open + write *)
		X.ADD_COM := 00;
	ELSE
		X.UCB.D_HEAD := WORD#16#F301; (* Filemode create + write *)
		X.ADD_COM := 02; (* ADD HEADER *)
	END_IF;

	X.UCB.D_MODE := 1; (* Dateinamen als String ablegen *)
	UCB(DATA:=X.UCB); (* Daten eintragen *)
	step_1 := 30;

30:	(* LOG-Trigger verarbeiten *)
	trig_tmp := (TRIG_M AND NOT trig_m_last) OR trig_auto OR X.ADD_DATA_REQ;

	IF ENABLE = FALSE OR fn <> fn_last THEN (* ENABLE = 0 oder neuen Dateinamen -> Log Stop *)
		trig_stored := trig_tmp; (* aktuellen Triggerpuls speichern *)
		X.UCB.D_HEAD := WORD#16#EE00;
		X.UCB.D_MODE := 1;
		UCB(DATA:=X.UCB); (* Element schreiben *)
		X.ADD_COM := 00;
		step_1 := 00;

		(* ---------------- Debug-Message -----------------------*)
		(*IF _debug_enable THEN
			LOG_CL.NEW_MSG := 'FILE_XML1 - Stop: [~2]';
			LOG_CL.PRINTF[2] := DT_TO_STRING(DTI);
			LOG_MSG();
		END_IF;*)
		(* -----------------------------------------------------------------*)

	ELSIF ENABLE THEN
		IF trig_tmp OR trig_stored THEN (* manueller, automatischer oder externer Trigger *)
			trig_stored := FALSE;
			X.ADD_COM := 03; (* ADD DATA *)
			SAVE_DATA.TRIG_CNT := SAVE_DATA.TRIG_CNT + UDINT#1;
			SAVE_DATA.TRIG_CNT_TOTAL  := SAVE_DATA.TRIG_CNT_TOTAL + UDINT#1;
			(* ---------------- Debug-Message -----------------------*)
			(*IF _debug_enable THEN
				LOG_CL.NEW_MSG := 'FILE_XML1 - Trig: [~2]';
				LOG_CL.PRINTF[2] := DT_TO_STRING(DTI);
				LOG_MSG();
			END_IF;*)
			(* -----------------------------------------------------------------*)
		ELSE
			X.ADD_COM := 04;	(* ADD DATA REQ *)
		END_IF;
	END_IF;

END_CASE;
X.ADD_DATA_REQ := FALSE; (* externe Anforderung rücksetzen *)

(* ##################################### *)

CASE step_2 OF

00:	aw_ton(IN:= idx > 0 AND aw_enable , PT:= AUTO_CLOSE); (* AutoWrite Timer *)
	IF aw_ton.Q THEN (* Zeitgesteuertes Datenschreiben *)
		aw_aktiv := TRUE;
		step_2 := 10; (* Daten schreiben *)
		(* ---------------- Debug-Message -----------------------*)
		(*IF _debug_enable THEN
			LOG_CL.NEW_MSG := 'FILE_XML2 - AutoWrite: [~2]';
			LOG_CL.PRINTF[2] := DT_TO_STRING(DTI);
			LOG_MSG();
		END_IF;*)
		(* -----------------------------------------------------------------*)

	ELSE
		wd_ton(IN:= FALSE, PT:= wd_time);
		wd_ton(IN:= TRUE);
		WHILE X.UCB.BUF_COUNT > 0 AND step_2 = 0 AND wd_ton.Q = FALSE DO

			X.UCB.D_MODE := 10;
			UCB(DATA:=X.UCB); (* Element lesen , aber noch nicht entfernen *)

			IF X.UCB.D_HEAD > WORD#16#F000 THEN (* F301 oder F201 *)

				str := '<?xml version="1.0" encoding="UTF-8"?><table>';

				IF idx + LEN(str) < SIZEOF(PT.BUFFER) THEN (* Platz für Element vorhanden ? *)

					FSD.MODE := WORD_TO_BYTE(SHR(SHL(X.UCB.D_HEAD,4),12)); (* 0X00 -> 000X = 3 create + write / 2 open + write *)
					FSD.OFFSET := UDINT#0; (* Start bei Dateianfang *)
					FSD.FILENAME := X.UCB.D_STRING; (* Dateiname *)
					PT.SIZE := UINT#0;
					SAVE_DATA.FN_REM := FSD.FILENAME; (* aktuellen Dateinamen remanent sichern *)

					X.NEW_FILE := FSD.FILENAME;
					X.NEW_FILE_SIZE := UDINT#0;
					X.NEW_FILE_RTRIG := FALSE;
					step_2 := 20;
	
					(* Headerdaten schreiben *)
					IF FSD.MODE = BYTE#3 THEN
						SAVE_DATA.TRIG_CNT := UDINT#0; (* Datei neu anlegen -> dann zähler reset *)

						OSCAT_BASIC._STRING_TO_BUFFER(STR:=str, POS:=idx, PT:=ADR(PT.BUFFER), SIZE:=SIZEOF(PT.BUFFER));
						idx := idx + LEN(str);
						X.NEW_FILE_SIZE := total_bytes + INT_TO_UDINT(idx);
					END_IF;

					X.UCB.D_MODE := 11;
					UCB(DATA:=X.UCB); (* Element entfernen *)

					(* ---------------- Debug-Message -----------------------*)
					(*IF _debug_enable THEN
						LOG_CL.NEW_MSG := 'FILE_XML2 - Create: Mode [~1] , [~2]';
						LOG_CL.PRINTF[2] := DT_TO_STRING(DTI);
						LOG_CL.PRINTF[1] := BYTE_TO_STRING(FSD.MODE);
						LOG_MSG();
					END_IF;*)
					(* -----------------------------------------------------------------*)
				END_IF;

			ELSIF X.UCB.D_HEAD = WORD#16#EE00 THEN (* LOG_STOP Command *)

				str := '</table>';

				IF idx + LEN(str) < SIZEOF(PT.BUFFER) THEN (* Platz für Element vorhanden ? *)

					OSCAT_BASIC._STRING_TO_BUFFER(STR:=str, POS:=idx, PT:=ADR(PT.BUFFER), SIZE:=SIZEOF(PT.BUFFER));
					idx := idx + LEN(str);
					log_stop := TRUE;
					step_2 := 10; (* Daten schreiben *)

					X.UCB.D_MODE := 11;
					UCB(DATA:=X.UCB); (* Element entfernen *)

				END_IF;

			ELSIF idx + LEN(X.UCB.D_STRING) + 120 < SIZEOF(PT.BUFFER) THEN (* Platz für Element vorhanden ? *)

				(* ---------------- Debug-Message -----------------------*)
				(*IF _debug_enable THEN
					LOG_CL.NEW_MSG := 'FILE_XML2 - BUF: TXT [~1],Pos [~2], [~3]';
					LOG_CL.PRINTF[1] := X.UCB.D_STRING;
					LOG_CL.PRINTF[2] := INT_TO_STRING(idx);
					LOG_CL.PRINTF[3] := DT_TO_STRING(DTI);
					LOG_MSG();
				END_IF;*)
				(* -----------------------------------------------------------------*)

				IF log_state = USINT#0 THEN
					str := '<row><entry>';
				ELSE
					str := '<entry>';
				END_IF;

				OSCAT_BASIC._STRING_TO_BUFFER(STR:=str, POS:=idx, PT:=ADR(PT.BUFFER), SIZE:=SIZEOF(PT.BUFFER));
				idx := idx + LEN(str);
				log_state := log_state + USINT#1;

				OSCAT_BASIC._STRING_TO_BUFFER(STR:=X.UCB.D_STRING, POS:=idx, PT:=ADR(PT.BUFFER), SIZE:=SIZEOF(PT.BUFFER));
				idx := idx + LEN(X.UCB.D_STRING);

				n := n + USINT#1;
				IF n >= X.ID_MAX THEN
					n := USINT#0;
					str := '</entry></row>';
					log_state := USINT#0;
				ELSE
					str := '</entry>';
				END_IF;
				OSCAT_BASIC._STRING_TO_BUFFER(STR:=str, POS:=idx, PT:=ADR(PT.BUFFER), SIZE:=SIZEOF(PT.BUFFER));
				idx := idx + LEN(str);
				X.NEW_FILE_SIZE := total_bytes + INT_TO_UDINT(idx);

				X.UCB.D_MODE := 11;
				UCB(DATA:=X.UCB); (* Element entfernen *)

			ELSE (* kein Platz vorhanden *)
				step_2 := 10; (* Daten schreiben *)
			END_IF;
			wd_ton();
		END_WHILE;
	END_IF;

10:	IF idx > 0 THEN (* Daten schreiben *)
		FSD.MODE := BYTE#2; (* File_Open_Exist + File_Write *)
		FSD.OFFSET := UDINT#4294967294; (* 16#FFFF_FFFE ->Spezialcode: Daten automatisch an Dateiende anhängen *)
		PT.SIZE := INT_TO_UINT(idx); (* Datenlänge eintragen *)
		idx := 0;
		(* ---------------- Debug-Message -----------------------*)
		(*IF _debug_enable THEN
			LOG_CL.NEW_MSG := 'FILE_XML2 - WriteData: Mode [~3] Size [~1] , [~2]';
			LOG_CL.PRINTF[1] := UINT_TO_STRING(PT.SIZE);
			LOG_CL.PRINTF[2] := DT_TO_STRING(DTI);
			LOG_CL.PRINTF[3] := BYTE_TO_STRING(FSD.MODE);
			LOG_MSG();
		END_IF;*)
		(* -----------------------------------------------------------------*)
	END_IF;
	step_2 := 20;

